# B&R Automation Studio project TD52 (part 126)

### Module_IC.var - Module global variables
```iecst
VAR
	ucEnergLev : USINT; (* ignition system energy level % *)
	ActTiming : INT; (* actual ignition timing 1/10 degree *)
	AdvTimLi : INT; (* advanced ingnition timing 1/10 deg *)
	AnzSPnt : USINT; (* number of ignition speed points *)
	AvgTim : SINT; (* average ignition timing 1/10 deg. *)
	bGnlTrip : BOOL;
	bGnlTrip1 : BOOL;
	bGnlTrip2 : BOOL;
	bGnlTrip3 : BOOL;
	bGnlWarning : BOOL;
	bInitOK : BOOL;
	bSelfTestOn : BOOL; (* TRUE= ignition is in sleftest mode *)
	bSpeedTrig2 : BOOL; (* TRUE=inverse speed trig 2 output *)
	BWS_HA : BOOL := 0; (* Betriebswahlschalter Hand/Auto *)
	CMSIgn_Init : CMSinit;
	CMSmain_Ign : CMSmain;
	ConfigIC : USINT; (* ignition system operating mode *)
	EnergLev : USINT; (* ignition system energy level in % *)
	E_Conf : ARRAY[0..38] OF USINT; (* event ignition system parameter *)
	E_IgnErr : USINT; (* events igniton system error *)
	E_IgnHW : USINT; (* events ignition system hardware *)
	E_IgnStat : USINT; (* events igniton system status *)
	E_Missf : ARRAY[0..2] OF USINT; (* events for misfire control *)
	E_SpeedUpd : USINT; (* event for ign. speed update time *)
	E_Timing : ARRAY[0..24] OF USINT; (* events ign. syetem indiv. timing *)
	E_ZDGSpeed : USINT; (* events for ignition engine speed *)
	FGDRPS : BOOL; (* Freigabe durch RPS *)
	FireOrder : ARRAY[0..24] OF USINT; (* engine ignition fire order *)
	GloTiPnt : INT; (* global timing point 1/10 degree *)
	GoSelftest : BOOL; (* switch ignition system to selftest *)
	ic900_vis : BOOL; (* TRUE=CAN ignition system is used *)
	iCylCount : USINT; (*Loop counter*)
	IC_Node : USINT; (* ignition system node number *)
	iECanDevGo : DINT;
	IgnErr : ARRAY[0..7] OF USINT; (* ignition system error messages *)
	IgnHW : ARRAY[0..7] OF USINT; (* ignition system hardware info *)
	IgnOFail : ARRAY[0..24] OF BOOL; (* ignition system cyl.output failure *)
	IgnStat : ARRAY[0..6] OF USINT; (* ignition system status info *)
	IgnVers : UINT; (* ignition system software version *)
	IndivTim : ARRAY[0..24] OF SINT; (* cylinder individual timing offset *)
	IN_IC : IN_IC_Struct := (0);
	MissfCmd : BOOL; (* command for start misfire *)
	MissfCyl : UDINT; (* cylinder misfire parameter *)
	MissfTim : UINT; (* misfire time parameter *)
	MM2VIS : MM2VIS_Struct;
	ModeIC : USINT; (* ignition system operating mode *)
	M_AGFD : BOOL := 0; (* Aggregat angefordert *)
	n_ist : INT; (* actual speed [1/min] *)
	OutFailR : USINT; (* ignition output failure rate para. *)
	OUT_IC : OUT_IC_Struct := (0);
	OvrSpeed : UINT; (* ignition overspeed parameter *)
	Para : PARA_IC_Struct;
	ParaFactoryDefault : PARA_IC_Struct := (0);
	pm : PARA_IC_Struct;
	PosResetIC : INT; (* ignition reset pickup position *)
	PROBE : BOOL := 0; (* Betriebsart PROBE *)
	QUITTRPS : BOOL := 0; (* ack comand to PLC-part *)
	RetTimLi : INT; (* ignition retard timing limit *)
	SecSpeed : UINT; (* ignition system security speed *)
	SecSpeedOld : UINT; (* last security speed value *)
	SpeedHys1 : UINT; (* hysteresis ign. speed trigger 1 *)
	SpeedHys2 : UINT; (* hysteresis ign. speed trigger 2 *)
	SpeedPnt : ARRAY[0..4] OF UINT; (* ignition timing speed points *)
	SpeedTrg2 : INT; (* ignition system speed trigger 2 *)
	SpeedTrig1 : INT; (* ignition system speed trigger 1 *)
	SpeedTrig2 : INT; (* ignition system speed trigger 2 *)
	SpeedUpd : UINT; (* ignition speed update time [ms] *)
	StopM : BOOL; (* TRUE=engine is stopped *)
	TimeSPnt : ARRAY[0..4] OF INT; (* ignition speed point timing *)
	TimingSeq : USINT; (* ignition system timing sequence *)
	ucIC900CommErrCount : USINT; (* comm. error counter *)
	ucIgnType : USINT; (* ignition system hardware type *)
	ucOutpFRate : USINT; (* ignition output failure rate para. *)
	ucZuendabst : USINT; (* ignition timing diff. row A to B *)
	ucZylZAus : USINT; (* cyl.inder with output failure *)
	usActSpeed : UINT; (* actual engine speed by ignition *)
	usIgnSystem : UINT; (* hardware type of ignition system *)
	usZahnzahl : UINT; (* number of starter ring gear teeth *)
	W_ZZP : INT; (* actual ignition timing setpoint *)
	xEngtype : EngType; (*FB for engine type specific values*)
	xOpMode : OpMode; (*FB for engine operation mode*)
	ZDGAUS : ARRAY[0..24] OF BOOL := [25(0)]; (*Ignition output monitoring*)
	ZDGAUS_A : BOOL; (*Ignition output monitoring*)
	ZDGAUS_B : BOOL; (*Ignition output monitoring*)
	ZDGAUS_W : BOOL; (*Ignition output monitoring*)
	ZDGCAM : BOOL := 0; (* ZDG AUSFALL CAM PICKUP *)
	ZDGCAN : BOOL := 0; (*Ignition CAN communication failure*)
	ZDGCPU : BOOL := 0; (* ZDG CPU FEHLER *)
	ZDGFALSCH : BOOL := 0; (*Wrong type of ignition system*)
	ZDGPAR : BOOL := 0; (* ZDG PARAMETRIERUNG IM BETRIEB *)
	ZDGPARAM : BOOL := 0; (* ZDG PARAMETER FEHLER *)
	ZDGRST : BOOL := 0; (* ZDG AUSFALL RESET PICKUP *)
	ZDGSpeed : tZDGSpeed; (* engine speed meassured by ignition *)
	ZDGTRI : BOOL := 0; (* ZDG AUSFALL TRIGGER PICKUP *)
	ZDGUEDZ : BOOL := 0; (*Ignition shutoff overspeed*)
	ZUEND : BOOL := 0; (*Ignition on*)
	ZylZahl : USINT;
	ZZPAvg : INT; (* actual ignition point average *)
	ZZPCyl : ARRAY[0..24] OF INT; (* actual cylinder igniton point *)
	ZZPMax : INT; (* actual max.cylinder ignition point *)
	ZZPMin : INT; (* actual min.cylinder ignition point *)
	zzp_ist : INT; (* aktuelle Soll-ZZP ohne Reduktion *)
	bNoInitDetected : BOOL := FALSE; (*allways true, except 1cycle on init up*)
	CMSmainTrigger : BOOL := FALSE; (*Trigger variable for CMS_main()*)
	SIM_rN_IgnIC_Act : REAL; (*WINMOD simulation: Engine speed measured by ignition IC*)
	iNum_ICSys : USINT; (*IC-System*)
	tIC_FiringDist : IC_FiringDist; (*Firing distances*)
	tIC_Curr : ARRAY[0..6] OF IC_Curr; (*Ignition pulse current and duration*)
	tIC_CoilPara : IC_CoilPara; (*General coil parameters*)
	tIC_SpDur : IC_SpDur; (*Spark duration*)
	tIC_SpdST : IC_SpdST; (*Self-test speed and speed ramp up / down time*)
	iTi_ICOn : UINT; (*Hours powered-up [h]*)
	tIC_U_Pickups : IC_U_Pickups; (*Pickup peak voltages*)
	iNum_PUMode : USINT; (*Pickup mode detected by SEMIC*)
	iNum_IC_SPAxSpdCoeff : UINT; (*SPAx speed coefficient A*)
	E_Global : ARRAY[0..21] OF USINT; (*Even variables for ignition global parameters*)
	tIC_SpInfo : ARRAY[0..24] OF IC_SpInfo; (*Spark voltage and primary energy demand*)
	E_IC_SpInfo : ARRAY[0..24] OF USINT; (*Event variables for spark voltage and primary energy demand*)
	iNum_IC_NrTeethErr : UINT; (*Number of teeth at pickup error*)
	E_IC_NrTeethErr : USINT; (*Event variable for number of teeth at pickup error*)
	iT_IC : INT; (*Ignition controller temperature [degC*10]*)
	E_T_IC : USINT; (*Event variable for ignition controller temperature*)
	iU_IC_Supply : INT; (*Ignition controller supply voltage [V*10]*)
	E_U_IC_Supply : USINT; (*Event variable for ignition controller supply voltage*)
	tIC_PUNoiseRate : IC_PUNoiseRate; (*Pickup noise rate*)
	E_IC_PUNoiseRate : USINT; (*Event variable for pickup noise rate*)
	tIC_PrimEnergyStat : IC_PrimEnergyStat; (*Minimum, maximum and average of the primary coil energy demand*)
	E_IC_PrimEnergyStat : USINT; (*Event variable for the minimum, maximum and average of the primary coil energy demand*)
	bB_TrigFail : BOOL; (*Operating message - Ignition failure trigger pickup*)
	bW_CamFail : BOOL; (*Warning - Ignition failure cam pickup*)
	bW_ResetFail : BOOL; (*Warning - Ignition failure reset pickup*)
	bW_TrigFail : BOOL; (*Warning - Ignition failure trigger pickup*)
	iNum_TrigFail : USINT; (*Operating message - Ignition failure trigger pickup - Indication*)
	tCoilParam : ARRAY[0..4] OF CoilParam; (*Coil parameters*)
	tCoilParam5 : CoilParam5; (*Coil parameters*)
	tCoilParam6 : CoilParam6; (*Coil parameters*)
	iNum_IC_Curr7 : UINT; (*Ignition pulse 7 current*)
	iTi_IC_IonTime : UINT; (*Ionization time [us]*)
	bW_IC_WrongFw : BOOL; (*Wrong ignition controller firmware*)
	iE_PrimEnergy_Min : UINT; (*Minimum primary energy demand [mJ]*)
	iE_PrimEnergy_Max : UINT; (*Maximum primary energy demand [mJ]*)
	iE_PrimEnergy_Avg : UINT; (*Average primary energy demand [mJ]*)
	bW_PUDegrad : BOOL; (*Warning - Pickup degradation*)
	VIS2MM : VIS2MM_Struct;
	bIC_BlockUpd : BOOL; (*Block engine stat during ignition controler firmware update*)
	bW_IC_Uin_Lo : BOOL; (*Warning - Ignition controller input voltage too low*)
	bA_IC_HwFail : BOOL; (*Alarm - Ignition controller hardware failure*)
	bSEMIC_Comm : BOOL; (*SEMIC CAN communication is active*)
	bW_PUWrongPol : BOOL; (*Wrong pickup polarity*)
	bA_WrongCoil : BOOL; (*Alarm - Wrong or missing ignition coil*)
	bB_WrongCoil : BOOL; (*Operating message - Wrong or missing ignition coil*)
	iNum_WrongCoil : USINT; (*Operating message - Wrong or missing ignition coil - Cylinder number*)
	bA_IC_CoilFail : BOOL; (*Alarm - Ignition coil or wiring failure*)
END_VAR
```

### Module_ICPara.typ - Module global parameter
```iecst
TYPE
	PROGRAMMER_INFO : 	STRUCT
		DO_NOT_SORT_PARA : STRING[40] := 'DO NOT CHANGE PARAMETER SORTING!'; (*DO NOT CHANGE PARAMETER SORTING!*) (*ADD NEW PARAMETER ONLY AT THE END OF THE Para STRUCTURE. DO NOT DELETE existing Para items.*)
	END_STRUCT;
	PARA_IC_Struct : 	STRUCT
		iEng_Motortype : INT; (*PARA: engine motortype*) (*OldName:motortyp; Cycle:;*)
		rCA_AdvTimeLim : REAL; (*PARA [12065]: advanced ignition timing 1/10 deg *) (*OldName:AdvTimLi; Cycle:;*)
		b_IgnIC_SpdTrig2Inv : BOOL; (*PARA [12053]: TRUE=inverse speed trig 2 output *) (*OldName:bSpeedTrig2; Cycle:;*)
		rIgnIC_PowLev : REAL; (*PARA [12056]: ignition system energy level in % *) (*OldName:EnergLev; Cycle:;*)
		b_IgnIC_900Active : BOOL; (*PARA [12062]: TRUE=CAN ignition system is used *) (*OldName:ic900_vis; Cycle:;*)
		r_IgnIC_OutpMon : REAL; (*PARA [12054]: ignition output failure rate para. *) (*OldName:OutFailR; Cycle:;*)
		rN_OvrSpeed : REAL; (*PARA [12129]: Ignition overspeed limit*) (*OldName:OvrSpeed; Cycle:;*)
		r_IgnIC_ResPosIC : REAL; (*PARA [12055]: ignition reset pickup position *) (*OldName:r_IgnIC_ResPosIC; Cycle:;*)
		rCA_RetTimeLim : REAL; (*PARA [12066]: ignition retard timing limit *) (*OldName:RetTimLi; Cycle:;*)
		rN_IgnIC_SecSpeed : REAL; (*PARA [12059]: ignition system security speed *) (*OldName:SecSpeed; Cycle:;*)
		rN_IgnIC_HySpeed1 : REAL; (*PARA [12057]: hysteresis ign. speed trigger 1 *) (*OldName:SpeedHys1; Cycle:;*)
		rN_IgnIC_HySpeed2 : REAL; (*PARA [12058]: hysteresis ign. speed trigger 2 *) (*OldName:SpeedHys2; Cycle:;*)
		rN_IgnIC_SpeedTrig1 : REAL; (*PARA [12060]: ignition system speed trigger 1 *) (*OldName:SpeedTrig1; Cycle:;*)
		rN_IgnIC_SpeedTrig2 : REAL; (*PARA [12061]: ignition system speed trigger 2 *) (*OldName:SpeedTrig2; Cycle:;*)
		zz_V4_0_ParaVersionEnd : REAL := 4.0; (*! ADD NEW PARAMETER ONLY BELOW THIS LINE ! This is the end of base version parameter and has to stay unchanged. DO NOT CHANGE SORT ORDER of Para!*) (* OldName: new PV; Cycle: 5; *)
		bSEMIC_Active : BOOL; (*PARA[14519]: Ignition controller SEMIC*)
		rNum_IC_RelFwVer : REAL; (*PARA[14520]: Released SEMIC firmware version*)
		iNum_IC_PUMode : USINT; (*PARA[14521]: Pickup mode*)
		iNum_IC_CoilType : USINT; (*PARA[14522]: SEMIC coil type*)
		iTi_IC_TimeToPeak : UINT; (*PARA[14523]: Time to peak voltage [us]*)
		iI_IC_CoilCurrMax : USINT; (*PARA[14524]: Maximum primary coil current [A]*)
		iNum_IC_IgnEnergyMax : UINT; (*PARA[14525]: Maximum energy for firing event [mJ]*)
		iSpd_IC_PUMon : UINT; (*PARA[14526]: Speed to activate pickup monitoring [rpm]*)
		rU_IC_PUMin : REAL; (*PARA[14527]: Minimum pickup voltage [V]*)
		rSA_SparkDuration : REAL; (*PARA [12152]: SAFI spark duration  *)
		rSA_DurTol : REAL; (*PARA [12134]: spark duration deviation limit *) (* OldName:ucDurTol; Cycle: *)
		rSA_SparkCurChar : REAL; (*PARA [12150]: spark current characteristic*)
		rSA_SparkCurLev : REAL; (*PARA [12151]: spark current level *) (* OldName:ucSparkCurLev; Cycle: *)
		bDynSparkDuration : BOOL; (*PARA [13646]: Variable spark duration active *) (* OldName:newPV; Cycle: *)
		rP_Act_DynSpark_Limit_Nom : REAL; (*PARA [13648]: Spark duration below power threshold *) (* OldName:newPV; Cycle: *)
		usDurationIdle : UINT; (*PARA [13647]: Spark duration below power threshold *) (* OldName:newPV; Cycle: *)
		tSA_Ign_0 : IC_CurrPmmReal; (*PARA [12165]: SAFI ionization duration*) (* OldName:SAFICurr0PMM; Cycle: *)
		tSA_Ign_1 : IC_CurrPmmReal; (*PARA [12166] & PARA [12167] SAFI ignition current / duration setting 1 *) (* OldName:SAFICurr1PMM; Cycle: *)
		tSA_Ign_2 : IC_CurrPmmReal; (*PARA [12168] & PARA [12169]: SAFI ignition current / duration setting 2 *) (* OldName:SAFICurr2PMM; Cycle: *)
		tSA_Ign_3 : IC_CurrPmmReal; (*PARA [12170] & PARA [12171]: SAFI ignition current / duration setting 3 *) (* OldName:SAFICurr3PMM; Cycle: *)
		tSA_Ign_4 : IC_CurrPmmReal; (*PARA [12172] & PARA [12173]: SAFI ignition current / duration setting 4 *) (* OldName:SAFICurr4PMM; Cycle: *)
		tSA_Ign_5 : IC_CurrPmmReal; (*PARA [12174] & PARA [12175]: SAFI ignition current / duration setting 5 *) (* OldName:SAFICurr5PMM; Cycle: *)
		tSA_Ign_6 : IC_CurrPmmReal; (*PARA [12176]: SAFI ignition current setting 6 *) (* OldName:SAFICurr6PMM; Cycle: *)
		rNum_IC_TPCSCx1 : REAL; (*PARA[14528]: Breakpoint of secondary current axis for the target primary current 2D-MAP - X1*)
		rNum_IC_TPCSCx2 : REAL; (*PARA[14529]: Breakpoint of secondary current axis for the target primary current 2D-MAP - X2*)
		rNum_IC_TPCSCx3 : REAL; (*PARA[14530]: Breakpoint of secondary current axis for the target primary current 2D-MAP - X3*)
		rNum_IC_TPCSCx4 : REAL; (*PARA[14531]: Breakpoint of secondary current axis for the target primary current 2D-MAP - X4*)
		iNum_IC_TPCAPVy1 : USINT; (*PARA[14532]: Breakpoint of accumulated primary voltage axis for the target primary current 2D-MAP - Y1*)
		iNum_IC_TPCAPVy2 : USINT; (*PARA[14533]: Breakpoint of accumulated primary voltage axis for the target primary current 2D-MAP - Y2*)
		iNum_IC_TPCAPVy3 : USINT; (*PARA[14534]: Breakpoint of accumulated primary voltage axis for the target primary current 2D-MAP - Y3*)
		iNum_IC_TPCAPVy4 : USINT; (*PARA[14535]: Breakpoint of accumulated primary voltage axis for the target primary current 2D-MAP - Y4*)
		iI_IC_TPCx1y1 : USINT; (*PARA[14536]: Target primary current 2D-MAP data point - X1Y1*)
		iI_IC_TPCx1y2 : USINT; (*PARA[14537]: Target primary current 2D-MAP data point - X1Y2*)
		iI_IC_TPCx1y3 : USINT; (*PARA[14538]: Target primary current 2D-MAP data point - X1Y3*)
		iI_IC_TPCx1y4 : USINT; (*PARA[14539]: Target primary current 2D-MAP data point - X1Y4*)
		iI_IC_TPCx2y1 : USINT; (*PARA[14540]: Target primary current 2D-MAP data point - X2Y1*)
		iI_IC_TPCx2y2 : USINT; (*PARA[14541]: Target primary current 2D-MAP data point - X2Y2*)
		iI_IC_TPCx2y3 : USINT; (*PARA[14542]: Target primary current 2D-MAP data point - X2Y3*)
		iI_IC_TPCx2y4 : USINT; (*PARA[14543]: Target primary current 2D-MAP data point - X2Y4*)
		iI_IC_TPCx3y1 : USINT; (*PARA[14544]: Target primary current 2D-MAP data point - X3Y1*)
		iI_IC_TPCx3y2 : USINT; (*PARA[14545]: Target primary current 2D-MAP data point - X3Y2*)
		iI_IC_TPCx3y3 : USINT; (*PARA[14546]: Target primary current 2D-MAP data point - X3Y3*)
		iI_IC_TPCx3y4 : USINT; (*PARA[14547]: Target primary current 2D-MAP data point - X3Y4*)
		iI_IC_TPCx4y1 : USINT; (*PARA[14548]: Target primary current 2D-MAP data point - X4Y1*)
		iI_IC_TPCx4y2 : USINT; (*PARA[14549]: Target primary current 2D-MAP data point - X4Y2*)
		iI_IC_TPCx4y3 : USINT; (*PARA[14550]: Target primary current 2D-MAP data point - X4Y3*)
		iI_IC_TPCx4y4 : USINT; (*PARA[14551]: Target primary current 2D-MAP data point - X4Y4*)
		rNum_IC_PVOTRPCx1 : REAL; (*PARA[14552]: Breakpoint of spark current axis for the primary voltage off time reference 1D-TABLE - X1*)
		rNum_IC_PVOTRPCx2 : REAL; (*PARA[14553]: Breakpoint of spark current axis for the primary voltage off time reference 1D-TABLE - X2*)
		rNum_IC_PVOTRPCx3 : REAL; (*PARA[14554]: Breakpoint of spark current axis for the primary voltage off time reference 1D-TABLE - X3*)
		rNum_IC_PVOTRPCx4 : REAL; (*PARA[14555]: Breakpoint of spark current axis for the primary voltage off time reference 1D-TABLE - X4*)
		rNum_IC_PVOTRPCx5 : REAL; (*PARA[14556]: Breakpoint of spark current axis for the primary voltage off time reference 1D-TABLE - X5*)
		rNum_IC_PVOTRx1 : REAL; (*PARA[14557]: Duty cycle reference 1D-TABLE data point - X1*)
		rNum_IC_PVOTRx2 : REAL; (*PARA[14558]: Duty cycle reference 1D-TABLE data point - X2*)
		rNum_IC_PVOTRx3 : REAL; (*PARA[14559]: Duty cycle reference 1D-TABLE data point- X3*)
		rNum_IC_PVOTRx4 : REAL; (*PARA[14560]: Duty cycle reference 1D-TABLE data point- X4*)
		rNum_IC_PVOTRx5 : REAL; (*PARA[14561]: Duty cycle reference 1D-TABLE data point- X5*)
		iNum_IC_APVCF : USINT; (*PARA[14562]: Accumulated primary voltage compensation factor. Used for target primary current compensation for non nominal secondary voltage*)
		iI_IC_MPCPVOff : USINT; (*PARA[14617]: Calibration parameter for spark diagnostics. Minimum primary current after 250us spark duration if no 80v is applied*)
		iI_IC_MPCPVOn : USINT; (*PARA[14618]: Calibration parameter for spark diagnostics. Minimum primary current after 250us spark duration if 80v is applied for 250us*)
	END_STRUCT;
END_TYPE
```

### Program Logical/ICxx/IN_IC (IEC, version 4.12.0) - + IN-Task

- IN_ICCyclic.st (not readable text: treated as protected, skipped)

#### IN_IC.var - Local variables
```iecst
VAR
	iNum_IC_SpCurChar : USINT; (*Spark characteristic selection*)
	iNum_IC_SpCurLvl : USINT; (*Spark current level [%]*)
	iNum_IC_SpCurCharOld : USINT; (*Old spark characteristic selection*)
	iNum_IC_SpCurData : ARRAY[0..10] OF UINT; (*Data from IC_Curr.dat*)
	xDatObjRead_ICxxCurr : DatObjRead; (*FuB to read the data from IC_Curr.dat*)
	tIC_CurrPMM : ARRAY[0..7] OF IC_Curr; (*Ignition pulse current and duration from the parameters*)
	xDatObjInfo_ICxxCurr : DatObjInfo; (*FuB to read the info from IC_Curr.dat*)
	xDatObjInfo_ICxxCoil : DatObjInfo; (*FuB to read the info from IC_Coil.dat*)
	xDatObjRead_ICxxCoil : DatObjRead; (*FuB to read the data from IC_Coil.dat*)
	iNum_IC_CoilType : USINT; (*Coil type*)
	iNum_IC_CoilTypeOld : USINT; (*Old coil type*)
	iNum_IC_SpCoilData : ARRAY[0..39] OF UINT; (*Data from IC_Coil.dat*)
END_VAR
```

### Program Logical/ICxx/OUT_IC (IEC, version 4.14.0) - + OUT-Task

- OUT_ICCyclic.st (not readable text: treated as protected, skipped)

#### OUT_IC.var
```iecst
VAR
	xTON_IgnEngergy_Hi : TON; (*Timer for warning maximum energy exceeded*)
END_VAR
```

### Program Logical/ICxx/ignition (IEC, version 4.13.0) - + Main igniton task 

- ignitionCyclic.st (not readable text: treated as protected, skipped)

- ignitionInit.st (not readable text: treated as protected, skipped)

#### ignition.var
```iecst
VAR
	ucStateOfPar : USINT; (* state of parameter transmission *)
	bIC900Comm : BOOL; (* TRUE=communication to ignition OK *)
	bIgnOK : BOOL; (* TRUE=ignition system is OK *)
	bIgnFire : BOOL; (* TRUE=ignition system is firing *)
	bSendIC900Par : BOOL; (* flag sending ignition parameter *)
	bSendRunPar : BOOL; (* falg sending igniton run parameter *)
	bSendRunParError : BOOL; (* TRUE=error send ignition run para. *)
	bSendIC900ParError : BOOL; (* TRUE=error send igniton parameter *)
	bResetIC900 : BOOL; (* flag for reseting ignition system *)
	bChangeBetrArt : BOOL; (* TRUE=change ignition operating mod *)
	bChangeBTRFailure : BOOL; (* TRUE=fault change operating mode *)
	ucIgnOFailTimer : ARRAY[0..24] OF USINT; (* ignition output failure timer *)
	ucZylCount : USINT; (* cylinder loop counter *)
	ucModeIC : USINT; (* igniton system operating mode *)
	ucTimingSeq : USINT; (* ingition system timing sequence *)
	ucResetState : USINT; (* state of igniton reset sequence *)
	ucIC900Hours : UINT; (* ignition system operating hours *)
	usZahnzahlOld : UINT; (* number of starter ring gear teeth *)
	usSelfTestOnTime : UINT; (* timer for selftest on time *)
	bIC900Off : BOOL; (* TRUE=stop comm. to ignition system *)
	ssZZPMin : INT; (* actual min. indiv. timing point *)
	ssZZPMax : INT; (* actual max. indiv. timing point *)
	TON_ZDGTRI : TON; (* delay error missing ring gear *)
	F_TRIG_ZUEND : F_TRIG; (* faling trigger ignition system on *)
	R_TRIG_EngQuitt : R_TRIG; (* FUB trigger alarm reset pushed *)
	R_TRIG_EngStop : R_TRIG; (* FUB trigger operating switch stop *)
	R_TRIG_EngDemand : R_TRIG; (* FUB trigger for engine demand *)
	ucStateOfChange : USINT; (* state of change operating mode *)
	TON_ZDGRST : TON; (* FUB delay reset signal missing *)
	TON_ZDGPARAM : TON; (* FUB delay no config at enabele run *)
	TON_ZDGCAM : TON; (* FUB delay camshaft signal missing *)
	TON_BTRTimeOut : TON; (* 1 sec. timeout for sending IC mode *)
	ucIgnParCount : USINT; (* parameter error counter *)
	ucStateIgnPar : USINT; (* state of ignition parameter send *)
	bSendIgnParError : BOOL; (* TRUE=error send ignition parameter *)
	ucIndivTimCnt : USINT; (* loop counter individual timing *)
	PosResetICOld : INT; (* last ignition reset pickup pos. *)
	OutFailROld : USINT; (* last ign. outp. faulure rate para. *)
	AdvTimLiOld : INT; (* lat advanced timing limit *)
	RetTimLiOld : INT; (* last retard timing limit *)
	OvrSpeedOld : UINT; (* last over speed value *)
	SpeedTrig1Old : INT; (* last speed trigger 1 value *)
	SpeedTrig2Old : INT; (* last speed trigger 2 value *)
	SpeedHys1Old : UINT; (* last speed hystersis 1 value *)
	SpeedHys2Old : UINT; (* last speed hystersis 2 value *)
	TON_SecondTick : TON; (* second tick TRUE for 0,1 sec. *)
	ucNrOfZDGAUS : USINT; (* number of ign. output failures *)
	AmmSeqZDGAUS : AmmSequence; (* FUB AmmSequence ign. output fail. *)
	bSEMIC_ICmode : BOOL; (*SEMIC in IC-mode*)
	bIC_PUmodeRead : BOOL; (*PU mode read at least once since the CAN communication was open*)
END_VAR
```

### Program Logical/ICxx/SpeedIC (IEC, version 4.13.0) - + Engine speed ignition system IC

- SpeedICCyclic.st (not readable text: treated as protected, skipped)

#### SpeedIC.var - Local variables
```iecst
VAR
	MissfCyl_Old : UDINT;
	bIC_MissfCmd_Old : BOOL; (*Command to start skip fire - old*)
	xTOF_MissfCmd : TOF; (*Delay to turn off the skip fire command*)
END_VAR
```

### Program Logical/ICxx/ICGen (IEC, version 4.14.0) - + Task for general issues 

- GeneralCyclic.st (not readable text: treated as protected, skipped)

### Program Logical/ICxx/SEMIC (IEC, version 4.14.0) - + SEMIC ignition task

- SEMICCyclic.st (not readable text: treated as protected, skipped)

- SEMICInit.st (not readable text: treated as protected, skipped)

#### SEMIC.var - Local variables
```iecst
VAR CONSTANT
	all : SINT := 127;
	none : SINT := -1;
END_VAR
VAR
	bAmmSeqClkP : BOOL; (*Clock for AmmSequence*)
	bIC_RE_EngStop : BOOL; (*Rising edge of engine stopped + 5 s*)
	bIC_RE_SwReset : BOOL; (*Rising edge of the alarm reset button at engine stand still*)
	bIN_WrongFw : BOOL; (*Input of timer for alarm Wrong ignition controller firmware*)
	bSEMIC_CfgNotAllow : BOOL; (*Configuration parameters tranfer not allowed if engine is running*)
	bSEMIC_IgnFire : BOOL; (*Ignition firing*)
	bSEMIC_IgnOK : BOOL; (*Ignition OK*)
	bSEMIC_OpBeforeCfg : BOOL; (*Send operation data before the configuration data*)
	bSEMIC_SelfTestStart : BOOL; (*Start self test procedure for SEMIC*)
	bSEMIC_SelfTestStop : BOOL; (*Stop self test procedure for SEMIC*)
	bSEMIC_SendAllOpData : BOOL; (*Trigger the sending of all operating data*)
	bSEMIC_SendConfig : BOOL; (*Activate sending of configuration data*)
	bSEMIC_SwReset : BOOL; (*Start the SW reset procedure*)
	bToggle : BOOL;
	iCA_AdvTimLiOld : INT; (*Old advance timing limit*)
	iCA_ITPCyl : ARRAY[0..24] OF INT; (*Cylinder-specific ignition timing point difference from the global timing point*)
	iCA_PosResetICOld : INT; (*Old reset position*)
	iCA_RetTimLiOld : INT; (*Old retard timing limit*)
	iE_PrimEnergy_Sum : UDINT; (*Sum used to calculate the average primary coil energy demand*)
	iNum_Cnt : USINT;
	iNum_ConfigPara : SINT; (*Number of the configuration data to be sent*)
	iNum_ConfState : USINT; (*State of the configuration data sending sequence*)
	iNum_CylCnt : USINT;
	iNum_EnergLevOld : USINT; (*Old energy level*)
	iNum_GlobalPara : USINT; (*Number of the operating data to be sent*)
	iNum_ICSysOld : USINT; (*Old IC-system*)
	iNum_IC_Curr7Old : UINT; (*Old ignition pulse 7 current*)
	iNum_IC_SPAxSpdCoeffOld : UINT; (*Old SPAx speed coefficient A*)
	iNum_OutFailROld : USINT; (*Old output failure rate*)
	iNum_ParaCnt : USINT;
	iNum_ReadVarCnt : USINT; (*Counter for the variable read requests sequencing*)
	iNum_ReSendCnt : USINT;
	iNum_ResetState : USINT;
	iNum_SelfTestState : USINT;
	iNum_StartComCnt : USINT;
	iNum_TimingSeqOld : USINT; (*Old timing sequence*)
	iNum_ZahnzahlOld : UINT; (*Old number of gear teeth*)
	iNum_ZylZahlOld : USINT; (*Old number of cylinders*)
	iN_ActSpeed : UINT; (*Actual speed*)
	iN_OvrSpeedOld : UINT; (*Old overspeed*)
	iN_SpeedHys1Old : UINT; (*Old hysteresis speed trigger 1*)
	iN_SpeedHys2Old : UINT; (*Old hysteresis speed trigger 2*)
	iN_SpeedTrig1Old : INT; (*Old speed trigger 1*)
	iN_SpeedTrig2Old : INT; (*Old speed trigger 2*)
	iTi_IC_IonTimeOld : UINT; (*Old ionization time*)
	iTi_MissfTimOld : UINT; (*Old maximum skip fire duration*)
	iTi_SpeedUpdOld : UINT; (*Old speed update time*)
	tCoilParam5Old : CoilParam5; (*Old coil parameters*)
	tCoilParam6Old : CoilParam6; (*Old coil parameters*)
	tCoilParamOld : ARRAY[0..4] OF CoilParam; (*Old coil parameters*)
	tIC_CoilParaOld : IC_CoilPara; (*Old general coil parameters*)
	tIC_CurrOld : ARRAY[0..6] OF IC_Curr; (*Old ignition pulse current and duration*)
	tIC_FiringDistOld : IC_FiringDist; (*Old firing distances*)
	tIC_SpdSTOld : IC_SpdST; (*Old self-test speed and speed ramp up/down time*)
	tIC_SpDurOld : IC_SpDur; (*Old spark duration*)
	xAmmSeqIgnOFail : AmmSequence; (*Alarm sequence for Ignition output monitoring*)
	xAmmSeqWrongCoil : AmmSequence; (*Alarm sequence for Wrong or missing ignition coil*)
	xTON_100msTick : TON; (*100ms based clock pulse*)
	xTON_bW_TrigFail : TON; (*Timer for Warning - Ignition failure trigger pickup*)
	xTON_ConfFail : TON; (*Timer for configuration state too long*)
	xTON_EngineStop : TON; (*Timer for SEMIC software reset*)
	xTON_IcNoOpState : TON; (*Timer for Ignition parameter error if engine is demanded and IC is not in operation state*)
	xTON_IC_WrongFw : TON; (*Timer for alarm Wrong ignition controller firmware*)
	xTON_IgnDemFall : TON; (*Falling edge of the ignition demand*)
	xTON_IgnDemRise : TON; (*Rising edge of the ignition demand*)
	xTON_ResetFail : TON; (*Timer for ignition controller software reset too long*)
	xTON_SecondTick : TON; (*1s based clock pulse*)
	xTON_ZDGCAM : TON; (*Timer for Ignition failure cam pickup*)
	xTON_ZDGPARAM : TON; (*Timer for re-parametrization because of parametrization failure*)
	xTON_ZDGRST : TON; (*Timer for Ignition failure reset pickup*)
	xTON_ZDGTRI : TON; (*Timer for Alarm - Ignition failure trigger pickup*)
	xTON_ZDGTRI_4PU : TON; (*Timer for Alarm - Ignition failure trigger pickup in 4-pickups mode*)
	xTON_ZDGTRI_NoFire : TON; (*Timer for Alarm - Ignition failure trigger pickup when ignition not firing*)
END_VAR
```

### Program Logical/ICxx/MsgIC (IEC, version 4.13.0) - + Messages

- MsgICCyclic.st (not readable text: treated as protected, skipped)

- MsgICInit.st (not readable text: treated as protected, skipped)

#### MsgIC.var - Local variables
```iecst
VAR
	iAdrAmmBase2MM : UDINT;
	iAdrMM2AmmBase : UDINT;
	xMsg3310 : Msg;
	xMsg3240 : Msg;
	xMsg3410 : Msg;
	xMsg3027 : Msg;
	xMsg3031 : Msg;
	xMsg3029 : Msg;
	xMsg3030 : Msg;
	xMsg3026 : Msg;
	xMsg3025 : Msg;
	xMsg3028 : Msg;
	xMsg3052 : Msg;
	xMsg3209 : Msg;
	xMsg9339 : Msg;
	xMsg9340 : Msg;
	xMsg9049 : Msg;
	xMsg9341 : Msg;
	xMsg9342 : Msg;
	xMsg9343 : Msg;
	xMsg9315 : Msg;
	xMsg2363 : Msg;
	xMsg2764 : Msg;
	xMsg2767 : Msg;
	xMsg2367 : Msg;
	xMsg9073 : Msg;
	xMsg2375 : Msg;
END_VAR
```

### Program Logical/ICxx/ParIC (IEC, version 4.06.0) - + Parameter handling

- perm_par.st (not readable text: treated as protected, skipped)

#### perm_par.var
```iecst
VAR
	tParaIntern : ParaHandler_typ; (*Connector type to perm_par*)
	tMM2ParaBase_ReadBack : MM2ParaBase_type; (*INTERNAL! V4.06 new readback structure for information from previous tasks*)
	bWriteDataObj : BOOL; (* TRUE=write data object module *)
	bDataObjLenErr : BOOL; (*Error occured in permem: data module size missmatch*)
	bCreateDataObj : BOOL; (* TRUE=create new data object *)
	bWriteOnce : BOOL; (* write permanent memory once *)
	DatObjCreate_01 : DatObjCreate; (* data object create *)
	DatObjInfoBak_02 : DatObjInfo; (* data object info *)
	DatObjDelete_01 : DatObjDelete; (* data object delete *)
	DatObjRead_01 : DatObjRead; (* data object read *)
	DatObjRead_02 : DatObjRead; (* manual initiated data object read *)
	DatObjWrite_01 : DatObjWrite; (* data object write *)
	DatObjDelete_02 : DatObjDelete; (* data object delete *)
	DatObjDelete_11 : DatObjDelete; (*Delete Backup File*)
	DatObjInfo_01 : DatObjInfo; (* data object info *)
	DatObjInfo_02 : DatObjInfo; (* data object info *)
	szModuleName : STRING[35]; (* module name of object *)
	szModuleNameBackup : STRING[35]; (* module name of posiibly created backup object *)
	DatObjCopy_01 : DatObjCopy;
	bCopyDataObj : BOOL;
	TON_WarnDelay : TON;
	TON_WritePMEM : TON; (* delay write permanent memory *)
	ulPMPointer : UDINT; (* adress of actual checksum value *)
	ulChecksum : UDINT; (* parameter checksum value *)
	pm_len : UDINT; (* permanent value lenght *)
	ulChecksumOld : UDINT; (* last vlaue of parameter checksum *)
	ulChkValue : UDINT; (* actual value of parameter pointer *)
	pm_id : UDINT; (* permanent value identifier *)
	pm_p : UDINT; (* permanent value pointer *)
	DatObjInfo_META : DatObjInfo;
	DatObjRead_META : DatObjRead;
	szMetaDataRaw : STRING[2000];
	szMetaData : ARRAY[0..4] OF STRING[35];
	szMetaDataVis : ARRAY[0..3] OF STRING[35];
	ssIndex : INT;
	ssCount : INT;
	ucMetaDataRaw : ARRAY[0..2000] OF USINT;
	ssCount2 : INT;
	szMetaDataFile : STRING[10];
	szText1 : STRING[20];
	pv_adr_IN_XX_tPB2MM : UDINT;
	pv_lng : UDINT;
	pv_lng_IN_XX_tPB2MM : UDINT;
	pv_lng_OUT_XX_tPB2MM : UDINT;
	szText2 : STRING[20];
	pv_adr_OUT_XX_tXX2PB : UDINT;
END_VAR
VAR CONSTANT
	ERR_NOERROR : UINT := 0;
END_VAR
VAR
	usPMWriteCnt : UINT;
	pm_Error : UDINT; (* permanent value error *) (* Deleted: pm : ParaMem_typ; permanent memory tags mathias, 22.8.11*)
	fun_Error : UDINT := 0; (*state > 0 = function error*)
	xLocalParaCheck : ParaCheckFUB; (*local function instance to check parameter values*)
	TON_ParaSetupOk : TON;
	bParaCheckSystemOk : BOOL;
	iDebug_ParaOkChecked : UDINT;
	bRestoreBackupDataObj : BOOL := FALSE;
	bRestoreDataObjContent : BOOL := FALSE;
	pm_id_backup : UDINT;
	pm_p_Backup : UDINT;
	DatObjCopy_02 : DatObjCopy;
	bDeleteBackupDataObj : BOOL := FALSE; (*Command to delete backup data module file on purpose*)
	bDebugPara : ARRAY[0..5] OF BOOL;
	ssIndex2 : INT;
	ssIndex3 : INT;
	ssIndex4 : INT;
	ssIndexVis : INT;
	szText : STRING[40];
	pv_adr_Para : UDINT;
	szParaSnippet : ARRAY[0..5] OF STRING[150];
	szParaIndex : STRING[10];
	slValue : DINT;
	iModuleDLD_ResetCount : INT;
	bDownloadDetected : BOOL;
	bFlagParaStructCopyWorking : BOOL; (*true, if cyclic para copying is active, 1 false cycle at every copy *)
	bStoreInitParaInDataObj : BOOL := FALSE;
	bTestflag : BOOL;
	bReadOutMETA_Once : BOOL;
	tParaCheck_iPvAdress : ARRAY[0..5] OF UDINT;
	tParaCheck_iPvLengt : ARRAY[0..5] OF UDINT;
	tParaCheck_rPvValue : ARRAY[0..5] OF REAL;
	tParaCheck_rRangeMIN : ARRAY[0..5] OF REAL;
	tParaCheck_rRangeMAX : ARRAY[0..5] OF REAL;
	tParaCheck_szPvName : ARRAY[0..5] OF STRING[35];
	ssFormatDetected : INT;
	szMetaDataPart : STRING[150];
	szFullTaskName : STRING[35];
	szFullMetaModuleName : STRING[35];
	debugLen : INT;
	debugSize : INT := 0;
	strcat_adr1 : UDINT;
	strcat_adr2 : UDINT;
	ssIndexTN : INT;
	bAlternate : BOOL;
	n : INT;
	iAlternateChecksum : DINT;
	iAlternateChecksumOld : DINT;
	ulDebugChkValue : ARRAY[0..999] OF UDINT;
	Adr1 : UDINT;
	Adr2 : UDINT;
	usPMWriteCntStepsize : UINT := 1; (*different step sizes to help debug*)
	usPMWriteCntXOR : UINT;
	usPMWriteCntAltSum : UINT;
	ulAdrPM : UDINT;
	usChkValuePM : USINT;
	ulAdrPara : UDINT;
	ulPara_len : UDINT;
	usChkValuePara : USINT;
	iDebugCountPMDifferences : DINT := 0;
	bEngineRunDetected : BOOL; (*detection status bit autocommand 100 /101  for engine run state*)
	ucMetaDataDebugInfoLine : ARRAY[0..24] OF STRING[80];
	ssIndexMand : INT := 0;
	szMetaDataMand : STRING[35];
	iMyErrorInfo_Autoreset : DINT; (*internal autoreset counter*)
	ssIndex_Version : INT; (*internal*)
	ssIndex_BU : INT; (*internal*)
	ssIndex_BU2 : INT; (*internal*)
END_VAR
```

### Program Logical/ICxx/VisIC (IEC, version 4.12.0) - + Visualization task

- VisICCyclic.st (not readable text: treated as protected, skipped)

#### VisIC.var - Local variables
```iecst
VAR
	iNum_CylCnt : USINT;
END_VAR
```

### Package Logical/ICxx/CAN - CAN communication IC

### Program Logical/ICxx/CAN/caniniIc (IEC, version 4.00.3) - + IC CAN communication init

#### caniniIcCyclic.st
```iecst
(*******************************************************************************
AGGR: intiate CAN communication (cyclic)

This code is confidential and proprietary to the INNIO Company.
It may not be used in any form, or reproduced in any manner, without the express
written permission of the INNIO Company.
Copyright, INNIO Company, 2022

Customized modifications: -
------------------------

History:
-------
V0.1		31-08-2001	Fahringer, generated from caninit.c V0.2
			31-08-2001	Fahringer, last modification
V0.21		14-10-2003	Weitzer,   transfer all CAN and CMS FUBs to caninit task
V0.40		14-02-2007  Weitzer,   change to new standard IF (SL1.SS1.IF2)
							   	   delete MMD (multimeasure device)
V0.50		07-09-2007	Weitzer,   SAFI added
							       main FUB´s moved to canmain program
V0.60		23-02-2010	Weitzer,   SAFI2 (prot injection) added
V4.00.03	10-07-2014	Denk,      AND ic900_vis added
V4.00.05	15-07-2015	Weitzer,   move CMS main Fub to SpeedIC task
V4.12.00	08-09-2022	Andre	   Select the engine speed from the ICxx module also if SEMIC is active

Instructions for use:
--------------------
-initiate the CAN-Bus communictation controller
-initiate CAN CMS manager

Outstandings:
------------
*******************************************************************************)

PROGRAM _CYCLIC

	IF IN_IC.iCANIdent <> 0 AND NOT bInitOK AND (ic900_vis OR Para.bSEMIC_Active) THEN	(* check if CAN open was successful *)

		(*initiate CMS manager Ignition *)
		CMSIgn_Init(enable:=1, us_ident:=IN_IC.iCANIdent, user_type:=0, queue_cnt:=0, modul_name:=ADR('cmsign'));
		(* initiate CMS main function for send and receive Ignition CAN messages *)
		CMSmain_Ign.enable    := TRUE;
		CMSmain_Ign.cms_ident := CMSIgn_Init.cms_ident;
		CMSmain_Ign.cms_mode  := 2;

		IF CMSIgn_Init.status = 0 THEN
			bInitOK := TRUE;
		END_IF
	END_IF

END_PROGRAM
```

### Data object Logical/ICxx/CAN/cmsign (Simple, version 4.12.0) - + IC CAL ignition

- cmsign.dat (binary file, 13439 bytes)
### Program Logical/ICxx/CAN/IC_Updater (IEC, version 4.13.0) - + IC CAN updater

- IC_UpdaterCyclic.st (not readable text: treated as protected, skipped)

- IC_UpdaterInit.st (not readable text: treated as protected, skipped)

#### IC_Updater.var - Local variables
```iecst
VAR
	bIC_StartFwUpd : BOOL; (*Start the IC firmware download*)
	CMSdlreq_IcFw : CMSdlreq; (*Function block to download IC firmware*)
	DatObjInfo_IcFw : DatObjInfo; (*Function block to get the info of the ICfirmware*)
	iNum_IcFwAdr : UDINT; (*IC firmware address*)
	iNum_IcFwLen : UDINT; (*IC firmware length*)
	iNum_IcFwStatus : UINT; (*IC firmware status*)
	iNum_IcUpdState : USINT;
	iNum_InitDlFwCnt : USINT; (*Counter to re-send the initiate domain download*)
	xTON_IC_Upd : TON; (*Limit the IC firmware download to 30 min*)
END_VAR
```

### Package Logical/ICxx/DataIC - Data ICxx

### Data object Logical/ICxx/DataIC/IC_Coil (Simple, version 4.12.0) - + IC coil type data

- IC_Coil.dat (binary file, 45687 bytes)
### Data object Logical/ICxx/DataIC/IC_Curr (Simple, version 4.12.0) - + IC spark current characteristic

- IC_Curr.dat (binary file, 12102 bytes)
### Package Logical/Ignition - IG: Ignition

### Data object Logical/Ignition/META_IG (Simple) - MODUL META data file

#### META_IG.dat
```
; *******************************************************************************
; AGGR: Module Meta Data (data module)
;
; This code is confidential and proprietary to the INNIO Company.
; It may not be used in any form, or reproduced in any manner, without the express
; written permission of the INNIO Company.
; Copyright, INNIO Company, 2025
;
; Customized modifications: -
; ------------------------
;
; History:
; -------
; V03.99.00.00	06.03.2013	Weitzer		generated for modular software
; V03.99.02.00	29.05.2013	Zengerer	initial dependencies prepared
; V04.00.00.00	30.01.2014	Denk		new version
; V04.01.00.00	22.07.2014	Denk		OUT_IG.rCA_Ign_Avg added, Para task updated, bIgn_SelfTest to MM2VIS added
; V04.03.00.00	02.11.2015	Zengerer 	MANDATORYMODULE statement
; V04.03.01.00	24.01.2018	Denk		bMsg1022, IN_IG.tPB2MM.bParaSetupOk added
; V04.07.00.00	23.01.2019	Zengerer	Distribute Para task with perm messaage handling capability to all modules, no functional change to V4.06
; V04.07.00.00	01.02.2019	Hohensinner	Ignition Information for custom module (bus applications)
; V04.09.00.00	10.12.2019	Denk		Ignition System Self-Test Improvements
; V04.11.00.00	22.12.2021	Andre		Use Para.bSA_Ign_Active to select ignition by SAFI or by MIC
; V04.12.00.00	08.09.2022	Andre		Select the engine speed from the ICxx module also if SEMIC is active
; V04.13.00.00	17.10.2023	Andre		Bugfix for M_STRDRE
;				05-12-2023	Bacci		Added ventilation demand and release before starting the self-test (2023-190)
;				05.03.2024	Bacci		Changes on trip 1061 added
; V04.14.00.00	27.11.2024	Andre		Display B3226 and prevent B3225 during purge starts with all cylinders skipped.
;				02.12.2024	Andre		Set ignition feedback from CAN to TRUE in simulation mode
;				13.02.2025	Andre		ZM2_ZEST not set while the early gas valve opening function is active.
;
; Instructions for use:
; --------------------
; make only changes at the version numbers
;
; Outstandings:
; ------------
;
; *******************************************************************************
;
"<META>"
;
; Module ID
"<MODUL>IG</MODUL>"
;
; Module Version (xx.yy.zz.cc)
"<VERSION>04.14.00.00</VERSION>"
;
; Module Basisupdate Version BU (00-99)
"<BASISUPDATE_VERSION>00</BASISUPDATE_VERSION>"
;
; Optional: specify order number for limitated module usage
"<ORDER></ORDER>" ;<!--(optional for restricted customizations; missing statement makes module valid for all orders)-->
;
; Parameter Check <PARAn Name='aAbcdef' MIN='xxx' MAX='yyy' />  (watch for correct spacings and apostrophs!)
"<PARAMETER_CHK>"
"	<PARA1 Name='iEng_Motortype' MIN='208' MAX='920' />"
"	<PARA2 />"
"	<PARA3 />"
"	<PARA4 />"
"	<PARA5 />"
"</PARAMETER_CHK>"
;
; Statement, if engine operation is also allowed without this module (FALSE) or if this module´s parameter check passing is mandatory (TRUE)
"<MANDATORYMODULE>TRUE</MANDATORYMODULE>"
;
; Permanent Datamodule Filenames<!-- enter filenames for counter and INTERNAL parameter only; filename without extention-->
"<DATAMODULES>" ;<!-- optional; mehrere DATAMODULES erlaubt-->
"	<DATAMODULE>par_IG</DATAMODULE>"
"</DATAMODULES>"
;
; Dependencies Modules (MMxx.yy.zz.cc)
"<DEPENDENCIES>"
"	<DEPENDENCY MODULE='SY' VERSION='04.00.00.00' />"
"	<DEPENDENCY MODULE='PB' VERSION='04.00.00.00' />"
"	<DEPENDENCY MODULE='SA' VERSION='04.00.00.00' />"
"	<DEPENDENCY MODULE='OP' VERSION='04.00.00.00' />"
"	<DEPENDENCY MODULE='MO' VERSION='04.00.00.00' />"
"	<DEPENDENCY MODULE='IC' VERSION='04.13.00.00' />"
"	<DEPENDENCY MODULE='HA' VERSION='04.13.00.00' />"
"	<DEPENDENCY MODULE='GT' VERSION='04.00.00.00' />"
"	<DEPENDENCY MODULE='EG' VERSION='04.00.00.00' />"
"	<DEPENDENCY MODULE='EC' VERSION='04.00.00.00' />"
"	<DEPENDENCY MODULE='AG' VERSION='04.14.00.00' />"
"	<DEPENDENCY MODULE='AB' VERSION='04.00.00.00' />"
"	<DEPENDENCY MODULE='GC' VERSION='04.03.00.00' />"
"	<DEPENDENCY MODULE='VE' VERSION='04.13.00.00' />"
"   <DEPENDENCY VISVERSION='02.12.03.00' />"			; Dependencies Visualization
"</DEPENDENCIES>"
;
; Module function description
"<MODULEFUNCTION>" ;<!-- short overview documentation of module function; add reference to detailed information, if available-->
"	<General>	"
"	 Handling of general ignition topics	"
"	</General>	"
""
"	<F1 Name='Engine speed' LastModified='04.00.00.00'>"
"	Engine speed handling depending on used ignition system. 	"
"	</F1>"
"	<F2 Name='Ignition voltage calculations' LastModified='04.00.00.00'>"
"	 Calculation of min, max and avg values depending on used ignition system.	"
"	</F2>"
"	<F3 Name='Timing point calculation' LastModified='04.00.00.00'>"
"	 Calculation of ignition timing point min, max and avg values depending on used ignition system. "
"	</F3>"
"	<F4 Name='Ignition selftest' LastModified='04.00.00.00'>"
"	Ignition system selftest mode functionallity. "
"	</F4>"
"	<F5 Name='Double Ignition' LastModified='04.00.00.00'>"
"	Double ignition functionallity and building of variable bIgn_Run. "
"	</F5>"
""
"	<Info>"
"	V4.01.00	01-07-2014	Denk 	MM2VIS.bIgn_SelfTest added	"
"   V4.01.00	09.07.2014	Denk	OUT_IG.rCA_Ign_Avg := ZZPAvg; added  "
"   V4.05.00	21.12.2017	Denk	Bugfix, ignition self test with IC/MIC	  "
"	</Info>"
""
"	<Customized LastModified='4.0.0.0'>	"
"	- Nothing "
"	</Customized>	"
""
"</MODULEFUNCTION>"
;
"</META>"
```

### Module_IG.typ - Module global data types
```iecst
TYPE
	IN_IG_Struct : 	STRUCT
		tPB2MM : ParaBase2MM_type; (*Data exchange structure to ParaBase*) (*OldName:new PV; Cycle:5;*)
		tAB2IG : AmmBase2MM; (*AMM structure*) (*OldName:new PV; Cycle:2;*)
		tIgn_Run_Hal : HALioDi_Type; (*DI: Ignition system running*) (*OldName:ZIB;Cycle:2;*)
		tIgn2_Run_Hal : HALioDi_Type; (*DI: Ignition system double running*) (*OldName:ZIB2; Cycle:2;*)
		tGCB_RUC : HALioDo_Type; (*DO: Generator circuit breaker release under voltage coil*) (*OldName:A_USP; Cycle:2;*)
		tIgn_OverspeedRelay : HALioDi_Type; (*DI: Overspeed relay *) (*OldName:UEDZ; Cycle:5;*)
		tGCB_On : HALioDi_Type; (*DI: generator circuit breaker closed *) (*OldName:GCB_ON; Cycle:5;*)
		bIgnOperating : BOOL; (*SAFI ignition system running*) (*OldName:ZIB; Cycle:2;*)
		bMsg1026 : BOOL; (*shutdown failure*) (*OldName:M_ANSTAB; Cycle:2;*)
		bIgn_Dem : BOOL; (*demand ignition*) (*OldName:ZUEND; Cycle:2;*)
		bIgn_Dem_TC5 : BOOL; (*demand ignition*) (*OldName:ZUEND; Cycle:2;*)
		bGV_On : BOOL; (*Command open gas valves*) (*OldName:M_GASV; Cycle:2;*)
		bGV_On_TC2 : BOOL; (*Command open gas valves*) (*OldName:M_GASV; Cycle:2;*)
		rCA_IgnP_Set : REAL; (*global ignition timing set point*) (*OldName:W_ZZP ; Cycle:2;*)
		rCA_Ign_Act : ARRAY[0..24]OF REAL; (*actual ignition timing *) (*OldName:ActTiming; Cycle:2;*)
		rN_IgnIC_Act : REAL; (*engine speed meassured by ignition *) (*OldName:ZDGSpeed; Cycle:2;*)
		rN_IgnSAFI_Act : REAL; (* engine speed meassured by ignition *) (*OldName:ZDGSpeed; Cycle:2;*)
		bPr_EOP_Prelub1 : BOOL; (* Vorschmierdruck 1 Pumpe *) (*OldName:AN_VSD1; Cycle:5;*)
		b_IgnIC_SelfTestBack : BOOL; (* switch ignition system to selftest *) (*OldName:GoSelftest; Cycle:5;*)
		b_IgnSAFI_SelfTestBack : BOOL; (* switch ignition system to selftest *) (*OldName:GoSelftest; Cycle:5;*)
		rU_IgnSAFI_Cyl : ARRAY[0..24]OF REAL; (*ignition voltage for each cylinder SAFI*) (*OldName:V_Zyl; Cycle:2;*)
		rU_IgnMon_Cyl : ARRAY[0..24]OF REAL; (*ignition voltage for each cylinder Monic*) (*OldName:V_Zyl; Cycle:2;*)
		bEng_Dem : BOOL; (*module demanded*) (*OldName:M_AGFD; Cycle:2;*)
		bDeflagrationPrct : BOOL; (*Deflagration protection*) (*OldName:PUFF; Cycle:2;*)
		bMnsOk : BOOL; (*Mains ok *) (*OldName:NE_OK; Cycle:5;*)
		bPr_EOP_Prelub2 : BOOL; (*Prelubrication pressure 2 pumps*) (*OldName:AN_VSD2; Cycle:5;*)
		bRelEngTurn_OilSkid : BOOL; (*release engine barring gear (Durchdrehvorrichtung) from Oil Skid*) (*OldName:new pv;Cycle:5*)
		bEngOilLevel_Lo : BOOL; (* engine oil level low *) (*OldName:ZM_OMIN; Cycle:5*)
		tSafetyLoop_EmStop : HALioDi_Type; (*safety loop - emergency stop*) (*OldName: DI_SIS; Cycle: 5;*)
		tSafetyLoop_Eng : HALioDi_Type; (*safety loop - engine*) (*OldName: RUHE, DI_RUHE_TC1; Cycle: 5;*)
		bSimWinMOD_Active : BOOL; (*WinMode simulation active *) (* OldName:new PV; Cycle:5*)
		iIdx_OMSS : INT; (* inex of operation mode selector switch - 0..OFF, 1..MAN, 2..AUTO, 3..TEST, 4..SCAVENGING *) (*OldName:new PV;Cycle:5;*)
		bInLouRelVE : BOOL; (*inlet louvers open or not closed*)
		bIC_Ign_Run_CAN : BOOL; (*IC Output ignition active from CAN*)
		bTOF_HwBypassDigitalTwin : BOOL; (*Hardware bypass digital twin - T3 adaptive cranking time*)
		bMsg2295 : BOOL; (*engine room ventilation failure inlet air*)
		bMissfCyl_PurgeCrk : BOOL; (*skip fire all cylinders while purging*)
	END_STRUCT;
	OUT_IG_Struct : 	STRUCT
		tIG2PB : MM2ParaBase_type; (*Data exchange structure to ParaBase*) (*OldName:new PV; Cycle:5;*)
		tIG2AB : MM2AmmBase; (*AMM structure*) (*OldName:new PV; Cycle:5;*)
		rN_EngAct : REAL; (*Engine Speed (1/min)*) (*OldName:ZDGSpeed; Cycle:2;*)
		bEO_PrelubeDemIgn : BOOL; (*Demand Prelubricating from ignition*) (*OldName:PRELUBE_IgnST; Cycle:2;*)
		bIgn_SelfTest : BOOL; (*Switch ignition system to selftest *) (*OldName:GoSelftest; Cycle:5;*)
		b_ST_DemIgn : BOOL; (*Demand starter from ignition*) (*OldName:STARTER_IgnST; Cycle:5;*)
		rU_Ign_Cyl : ARRAY[0..24]OF REAL; (*Ignition voltage for each cylinder *) (*OldName:V_Zyl; Cycle:;*)
		rU_Ign_Max : REAL; (* Maximum Ignition voltage *) (*OldName:AvgVolt; Cycle:;*)
		bIgn_Run : BOOL; (*Ignition system is running*) (*OldName:ZIB; Cycle:2;*)
		bN_EngStartDrop : BOOL; (*Engine start-up speed drop down*) (*OldName:M_STRDRE; Cycle:2;*)
		bMsg1022 : BOOL; (*Message*) (*OldName:M_UEDZ; Cycle:5;*)
		bIgn2_Sel : BOOL; (*TRUE = Double ignition selected*) (*OldName:IIXZUEND; Cycle:2;*)
		bMsg1064 : BOOL; (*Message *) (*OldName:M_UEDZRP; Cycle:5;*)
		bMsg3561 : BOOL; (*	Message	*) (*OldName:bPv; Cycle:5;*)
		tCA_IgnP_Set : HALioAo_Type; (*AO: timing point*) (*OldName:ssZZPOutWE; Cycle:2;*)
		bSelfTestRunning : BOOL;
		rCA_Ign_Avg : REAL; (*Actual ignition point average*) (*OldName:ZZPAvg; Cycle:;*)
		rU_Ign_Avg : REAL; (* *) (*OldName:AvgVolt; Cycle:;*)
		rU_Ign_Min : REAL; (* *) (*OldName:MinVolt; Cycle:;*)
		rCA_Ign_Min : REAL; (*Actual min. cylinder ignition point*) (*OldName:ZZPMin; Cycle:;*)
		rCA_Ign_Max : REAL; (*Actual max. cylinder ignition point*) (*OldName:ZZPMax; Cycle:;*)
		iIdx_IgnSelfTest : INT; (*Number of shown picture regarding step of execution. 0 - 50 in steps of 10. Detailded description in every step where used.*) (*OldName:usP5xSelftestStep; Cycle:;*)
		bInLouDemIgn : BOOL; (*Inlet louver demand for ignition selftest*)
		bIgn_Run_CAN : BOOL; (*Ignition system is running - feedback from CAN*)
	END_STRUCT;
	Para_IG_Struct : 	STRUCT
		bIgnMon_Active : BOOL; (*PARA [12064]: TRUE = MONIC is enabled/active*) (*OldName:monic_vis; Cycle:;*)
		bSA_Active : BOOL; (*PARA [12114]: TRUE = SAFI is enabled/active*) (*OldName:bSA_Active; Cycle:;*)
		b_IgnIC_900Active : BOOL; (*PARA [12062]: TRUE = CAN ignition system is used *) (*OldName:ic900_vis; Cycle:;*)
		bSA_Ign_Active : BOOL; (*PARA [12117]: TRUE = SAFI ignition function is enabled/active*) (*OldName:bSAFIIgn_Act; Cycle:;*)
		bIgn2_Sel_Para : BOOL; (*PARA [12063]: Select double ignition*) (*OldName:sel_2ignition; Cycle:;*)
		rN_EngStart_HyHi : REAL; (*PARA [11295]: speed engine start limit high hysteresis*) (*OldName:HY_DREHZ; Cycle:;*)
		rN_EngStart_LimHi : REAL; (*PARA [11296]: speed engine start limit high*) (*OldName:GW_DREHZ; Cycle:;*)
		rN_EngStartMon_HyHi : REAL; (*PARA [12067]: speed engine start monitoring limit high hysteresis*) (*OldName:HY_STRDRE; Cycle:;*)
		rN_EngStartMon_LimHi : REAL; (*PARA [12068]: speed engine start monitoring limit high*) (*OldName:GW_STRDRE; Cycle:;*)
		iEng_Motortype : INT; (*PARA: Motortype of the engine*) (*OldName:motortyp; Cycle:;*)
		rCA_RetTimeLim : REAL; (*PARA [12066]: Retard ignition timing limit*) (*OldName:RetTimLi; Cycle:;*)
		rCA_AdvTimeLim : REAL; (*PARA [12065]: Advanced ignition timing limit*) (*OldName:AdvTimLi; Cycle:;*)
		rN_PLC_LimHi : REAL; (*PARA [12070]: Overspeed PLC limit *) (*OldName:GW_UEDZ; Cycle:;*)
		rN_PLC_HyHi : REAL; (*PARA [12069]: Overspeed PLC hysteresis *) (*OldName:HY_UEDZ; Cycle:;*)
		tiIgn_SelfTest : TIME; (*PARA [14432]: Ignition self test duration*) (*OldName:monic_vis; Cycle:;*)
		bSEMIC_Active : BOOL; (*PARA[14519]: Ignition controller SEMIC*)
	END_STRUCT;
	MM2VIS_Struct : 	STRUCT
		rCA_Ign_Act : ARRAY[0..24]OF REAL; (*actual cylinder ignition point*) (*OldName:ActTiming; Cycle:;*)
		rCA_Ign_Avg : REAL; (*Actual ignition point average*) (*OldName:ZZPAvg; Cycle:;*)
		rCA_Ign_Min : REAL; (*Actual min. cylinder ignition point*) (*OldName:ZZPMin; Cycle:;*)
		rCA_Ign_Max : REAL; (*Actual max. cylinder ignition point*) (*OldName:ZZPMax; Cycle:;*)
		iIdx_IgnSelfTest : INT; (*Number of shown picture regarding step of execution. 0 - 50 in steps of 10. Detailded description in every step where used.*) (*OldName:usP5xSelftestStep; Cycle:;*)
		rU_Ign_Cyl : ARRAY[0..24]OF REAL; (*ignition voltage for each cylinder *) (*OldName:V_Zyl; Cycle:;*)
		rU_Ign_Avg : REAL; (* *) (*OldName:AvgVolt; Cycle:;*)
		rU_Ign_Max : REAL; (* *) (*OldName:MaxVolt; Cycle:;*)
		rU_Ign_Min : REAL; (* *) (*OldName:MinVolt; Cycle:;*)
		bMsg3346 : BOOL; (* *) (*OldName:; Cycle:;*)
		bMsg3228 : BOOL; (* *) (*OldName:; Cycle:;*)
		bMsg3347 : BOOL; (* *) (*OldName:; Cycle:;*)
		bMsg1061 : BOOL; (* *) (*OldName:; Cycle:;*)
		bMsg3225 : BOOL; (* *) (*OldName:; Cycle:;*)
		bMsg3226 : BOOL; (* *) (*OldName:; Cycle:;*)
		bMsg1022 : BOOL; (* *) (*OldName:; Cycle:;*)
		bMsg1064 : BOOL; (* *) (*OldName:; Cycle:;*)
		bMsg3561 : BOOL; (* *) (*OldName:; Cycle:;*)
		rN_EngAct : REAL; (*Engine Speed (1/min)*) (*OldName:; Cycle:;*)
		bIgn_SelfTest : BOOL; (*Switch ignition system to selftest *) (*OldName:GoSelftest; Cycle:5;*)
		bMsg9044 : BOOL; (* *) (*OldName:; Cycle:;*)
	END_STRUCT;
	VIS2MM_Struct : 	STRUCT
		bIgn_SelfTestStart : BOOL; (*start self test button*) (*OldName:; Cycle:;*)
		bIgn_SelfTestStop : BOOL; (*stop self test button*) (*OldName:; Cycle:;*)
		bIgn_SelfTestPrep : BOOL; (*start preperation button*) (*OldName:; Cycle:;*)
		bIgn_SelfTestCancel : BOOL; (*cancel preperation button*) (*OldName:; Cycle:;*)
		bHVMaxValueAct : BOOL; (*Spark voltage maximum*) (*OldName:; Cycle:;*)
	END_STRUCT;
END_TYPE
```

### Module_IG.var - Module global variables
```iecst
VAR
	M_DREHZ : BOOL; (* Startdrehzahl *)
	AN_STRDRE : BOOL; (* Startdrehzahl *)
	bGnlTrip1_IG : BOOL;
	bGnlTrip2_IG : BOOL;
	bGnlTrip3_IG : BOOL;
	bGnlTrip_IG : BOOL;
	bGnlWarning_IG : BOOL;
	bMsg1061_Set : BOOL; (*Module global variable to set message 1061*)
	iIdx_IgnSelfTest : INT; (*Number of shown picture regarding step of execution. 0 - 50 in steps of 10. Detailded description in every step where used.*)
	IN_IG : IN_IG_Struct;
	MM2VIS : MM2VIS_Struct;
	M_STRDRE : BOOL; (*Engine speed fallen below starter speed *)
	OUT_IG : OUT_IG_Struct;
	Para : Para_IG_Struct;
	ParaFactoryDefault : Para_IG_Struct := (0);
	pm : Para_IG_Struct;
	rU_Ign_Avg : REAL; (*Average ignition voltage*)
	rU_Ign_Max : REAL; (*Maximum ignition voltage*)
	rU_Ign_Min : REAL; (*Minimum ignition voltage*)
	usP5xSelftestStep : UINT;
	VIS2MM : VIS2MM_Struct;
	xEngtype : EngType; (*FB for Engine type specific values*)
	ZEST_1 : BOOL := 0; (*Ignition 1 failure*)
	ZEST_2 : BOOL := 0; (*Ignition 2 failure*)
	ZM1_ZEST : BOOL; (*Ignition failure*)
	ZM2_ZEST : BOOL; (*Ignition failure*)
	ZZPAvg : REAL; (* actual ignition point average *)
	ZZPMax : REAL; (* actual max.cylinder ignition point *)
	ZZPMin : REAL; (* actual min.cylinder ignition point *)
	bNoInitDetected : BOOL := FALSE; (*allways true, except 1cycle on init up*)
END_VAR
```

### Program Logical/Ignition/IGGen (IEC, version 4.14.0) - + General task

- IgnGenCyclic.st (not readable text: treated as protected, skipped)

- IgnGenInit.st (not readable text: treated as protected, skipped)

#### IgnGen.var - Local variables
```iecst
VAR
	ucCylinderCount : USINT;
	rU_IgnSAFI_Cyl : ARRAY[0..24] OF REAL; (*ignition voltage SAFI system for each cylinder local variable*)
	rU_IgnMon_Cyl : ARRAY[0..24] OF REAL; (*ignition voltage IC system for each cylinder local variable*)
	xGR_MAXR_EngSpeed : GR_MAXR; (*Limit max for Engine speed*)
	xGR_MAXR_EngineStartSpeed : GR_MAXR;
	ucCylIndex : USINT;
	rU_Ign_Avg_Sum : REAL; (*Average ignition voltage Temporary*)
	TON_SecondTick1 : TON; (* CAN BUS FAHLER *)
	TON_SecondTick : TON; (* CAN BUS FAHLER *)
	rU_Ign_Calc : ARRAY[0..24] OF REAL; (*ignition for each cylinder local variable*)
	rZZPAvg : REAL;
	bIgn_SelfTest : BOOL;
END_VAR
```

### Program Logical/Ignition/2xzuend (IEC, version 4.11.0) - + Double ignition

- 2xzuendCyclic.st (not readable text: treated as protected, skipped)

- 2xzuendInit.st (not readable text: treated as protected, skipped)

#### 2xzuend.var - Local variables
```iecst
VAR
	xTONIgn1FaultDelay : TON; (*Ignition1 fault delay *)
	xTONIgn2FaultDelay : TON; (*Ignition 2 fault delay *)
END_VAR
```

### Program Logical/Ignition/Selftest (IEC, version 4.13.0) - + Ignition selftest

- Selftest.st (not readable text: treated as protected, skipped)

#### Selftest.typ
```iecst
TYPE
	trafficLight_typ : 	STRUCT
		usP5xLightRed : UINT; (*Color of the traffic light*)
		usP5xLightYellow : UINT; (*Color of the traffic light*)
		usP5xLightGreen : UINT; (*Color of the traffic light*)
	END_STRUCT;
	Cylinder : 	STRUCT
		Selection : UINT;
		Data : ARRAY[0..24]OF UINT;
		Cyl : ARRAY[0..24]OF CylVal;
	END_STRUCT;
	CylVal : 	STRUCT
		Exh_Temp : INT;
		Spark_IP : INT;
		Spark_HV : INT;
		Knock_Int : INT;
		Knock_mV : INT;
		Valve_mV : INT;
		Press_bar : INT;
	END_STRUCT;
	bargraphScal_typ : 	STRUCT
		scScalEndValue : ARRAY[0..1]OF SINT; (*Start of the right limit area*)
		scScalStartValue : ARRAY[0..1]OF SINT; (*End of the left limit area*)
		scScalMaxDatapoint : ARRAY[0..1]OF SINT; (*Maximum value of the scale area*)
		scScalMinDatapoint : ARRAY[0..1]OF SINT; (*Minimum value of the scale area*)
		scBarValue : SINT; (*Value of the bargraph*)
		tShowBar : showBarColor_typ; (*Structur to show the OK-Bar (green) or the ERROR-Bar (red)*)
	END_STRUCT;
	showBarColor_typ : 	STRUCT
		ucStatusBarAct : USINT; (* Statusdatapoint for the GREEN Avg. Bar *)
		ucStatusBarMax : USINT; (* Statusdatapoint for the RED Limit Max Bar *)
		ucStatusBarMin : USINT; (* Statusdatapoint for the BLUE Limit Min Bar *)
	END_STRUCT;
	bargraphLeftRight_typ : 	STRUCT
		ucBarLeft : USINT; (*Value of the left bargraph*)
		ucBarRight : USINT; (*Value of the right bargraph*)
		scLimitLeft : SINT; (* Limitvalue to the left side *)
		scLimitRight : SINT; (* Limitvalue to the right side *)
		tShowBar : showBarLeftRight_typ; (*Structur to show the OK-Bar (green) or the ERROR-Bar (red)*)
	END_STRUCT;
	showBarLeftRight_typ : 	STRUCT
		ucStatusBarLeftAct : USINT; (* Statusdatapoint for the GREEN Avg. Bar *)
		ucStatusBarRightAct : USINT; (* Statusdatapoint for the GREEN Avg. Bar *)
		ucStatusBarMax : USINT; (* Statusdatapoint for the RED Limit Max Bar *)
		ucStatusBarMin : USINT; (* Statusdatapoint for the BLUE Limit Min Bar *)
	END_STRUCT;
END_TYPE
```

#### Selftest.var
```iecst
VAR
	xTON_SelftestPrelubCancel : TON;
	xTON_SelftestStarterWait : TON;
	xTON_SelftestStarter : TON;
	xTON_SelftestWait : TON;
	xTON_SelftestText : TON;
	bIgn_SelfTestBack : BOOL; (* switch ignition system to selftest, feedback ON signal from ignition systems*)
	xTON_SelftestBack : TON;
	tiSelftestBack : TIME := T#2s;
	xTON_SelfTest_Duration : TON;
END_VAR
```

### Program Logical/Ignition/MsgIG (IEC, version 4.14.0) - + Messages

- MsgIGCyclic.st (not readable text: treated as protected, skipped)

- MsgIGInit.st (not readable text: treated as protected, skipped)

#### MsgIG.var - Local variables
```iecst
VAR
	GR_MAX_OvrSpd : GR_MAXR;
	xMsg3561 : Msg;
	iAdrAmmBase2MM : UDINT;
	iAdrMM2AmmBase : UDINT;
	xMsg1061 : Msg;
	xMsg1022 : Msg;
	xMsg1064 : Msg;
	xMsg3225 : Msg;
	xMsg3226 : Msg;
	xMsg3228 : Msg;
	xMsg3346 : Msg;
	xMsg3347 : Msg;
	TP_R_GridOK : TP_R;
	bOverspdPLC : BOOL;
	T76 : BOOL; (*Ignition failure*)
	xTONIgnFail : TON; (*Ignition failure *)
	xTON_OpenGV_Mon : TON;
	xMsg9044 : Msg;
	SR_M_STRDRE : SR;
END_VAR
```

### Program Logical/Ignition/VisIG (IEC, version 4.01.0) - + Visualization task

- VisIGCyclic.st (not readable text: treated as protected, skipped)

- VisIGInit.st (not readable text: treated as protected, skipped)

### Program Logical/Ignition/ParIG (IEC, version 4.06.0) - + Parameter handling

- perm_par.st (not readable text: treated as protected, skipped)

#### perm_par.var
```iecst
VAR
	tParaIntern : ParaHandler_typ; (*Connector type to perm_par*)
	tMM2ParaBase_ReadBack : MM2ParaBase_type; (*INTERNAL! V4.06 new readback structure for information from previous tasks*)
	bWriteDataObj : BOOL; (* TRUE=write data object module *)
	bDataObjLenErr : BOOL; (*Error occured in permem: data module size missmatch*)
	bCreateDataObj : BOOL; (* TRUE=create new data object *)
	bWriteOnce : BOOL; (* write permanent memory once *)
	DatObjCreate_01 : DatObjCreate; (* data object create *)
	DatObjInfoBak_02 : DatObjInfo; (* data object info *)
	DatObjDelete_01 : DatObjDelete; (* data object delete *)
	DatObjRead_01 : DatObjRead; (* data object read *)
	DatObjRead_02 : DatObjRead; (* manual initiated data object read *)
	DatObjWrite_01 : DatObjWrite; (* data object write *)
	DatObjDelete_02 : DatObjDelete; (* data object delete *)
	DatObjDelete_11 : DatObjDelete; (*Delete Backup File*)
	DatObjInfo_01 : DatObjInfo; (* data object info *)
	DatObjInfo_02 : DatObjInfo; (* data object info *)
	szModuleName : STRING[35]; (* module name of object *)
	szModuleNameBackup : STRING[35]; (* module name of posiibly created backup object *)
	DatObjCopy_01 : DatObjCopy;
	bCopyDataObj : BOOL;
	TON_WarnDelay : TON;
	TON_WritePMEM : TON; (* delay write permanent memory *)
	ulPMPointer : UDINT; (* adress of actual checksum value *)
	ulChecksum : UDINT; (* parameter checksum value *)
	pm_len : UDINT; (* permanent value lenght *)
	ulChecksumOld : UDINT; (* last vlaue of parameter checksum *)
	ulChkValue : UDINT; (* actual value of parameter pointer *)
	pm_id : UDINT; (* permanent value identifier *)
	pm_p : UDINT; (* permanent value pointer *)
	DatObjInfo_META : DatObjInfo;
	DatObjRead_META : DatObjRead;
	szMetaDataRaw : STRING[2000];
	szMetaData : ARRAY[0..4] OF STRING[35];
	szMetaDataVis : ARRAY[0..3] OF STRING[35];
	ssIndex : INT;
	ssCount : INT;
	ucMetaDataRaw : ARRAY[0..2000] OF USINT;
	ssCount2 : INT;
	szMetaDataFile : STRING[10];
	szText1 : STRING[20];
	pv_adr_IN_XX_tPB2MM : UDINT;
	pv_lng : UDINT;
	pv_lng_IN_XX_tPB2MM : UDINT;
	pv_lng_OUT_XX_tPB2MM : UDINT;
	szText2 : STRING[20];
	pv_adr_OUT_XX_tXX2PB : UDINT;
END_VAR
VAR CONSTANT
	ERR_NOERROR : UINT := 0;
END_VAR
VAR
	usPMWriteCnt : UINT;
	pm_Error : UDINT; (* permanent value error *) (* Deleted: pm : ParaMem_typ; permanent memory tags mathias, 22.8.11*)
	fun_Error : UDINT := 0; (*state > 0 = function error*)
	xLocalParaCheck : ParaCheckFUB; (*local function instance to check parameter values*)
	TON_ParaSetupOk : TON;
	bParaCheckSystemOk : BOOL;
	iDebug_ParaOkChecked : UDINT;
	bRestoreBackupDataObj : BOOL := FALSE;
	bRestoreDataObjContent : BOOL := FALSE;
	pm_id_backup : UDINT;
	pm_p_Backup : UDINT;
	DatObjCopy_02 : DatObjCopy;
	bDeleteBackupDataObj : BOOL := FALSE; (*Command to delete backup data module file on purpose*)
	bDebugPara : ARRAY[0..5] OF BOOL;
	ssIndex2 : INT;
	ssIndex3 : INT;
	ssIndex4 : INT;
	ssIndexVis : INT;
	szText : STRING[40];
	pv_adr_Para : UDINT;
	szParaSnippet : ARRAY[0..5] OF STRING[150];
	szParaIndex : STRING[10];
	slValue : DINT;
	iModuleDLD_ResetCount : INT;
	bDownloadDetected : BOOL;
	bFlagParaStructCopyWorking : BOOL; (*true, if cyclic para copying is active, 1 false cycle at every copy *)
	bStoreInitParaInDataObj : BOOL := FALSE;
	bTestflag : BOOL;
	bReadOutMETA_Once : BOOL;
	tParaCheck_iPvAdress : ARRAY[0..5] OF UDINT;
	tParaCheck_iPvLengt : ARRAY[0..5] OF UDINT;
	tParaCheck_rPvValue : ARRAY[0..5] OF REAL;
	tParaCheck_rRangeMIN : ARRAY[0..5] OF REAL;
	tParaCheck_rRangeMAX : ARRAY[0..5] OF REAL;
	tParaCheck_szPvName : ARRAY[0..5] OF STRING[35];
	ssFormatDetected : INT;
	szMetaDataPart : STRING[150];
	szFullTaskName : STRING[35];
	szFullMetaModuleName : STRING[35];
	debugLen : INT;
	debugSize : INT := 0;
	strcat_adr1 : UDINT;
	strcat_adr2 : UDINT;
	ssIndexTN : INT;
	bAlternate : BOOL;
	n : INT;
	iAlternateChecksum : DINT;
	iAlternateChecksumOld : DINT;
	ulDebugChkValue : ARRAY[0..999] OF UDINT;
	Adr1 : UDINT;
	Adr2 : UDINT;
	usPMWriteCntStepsize : UINT := 1; (*different step sizes to help debug*)
	usPMWriteCntXOR : UINT;
	usPMWriteCntAltSum : UINT;
	ulAdrPM : UDINT;
	usChkValuePM : USINT;
	ulAdrPara : UDINT;
	ulPara_len : UDINT;
	usChkValuePara : USINT;
	iDebugCountPMDifferences : DINT := 0;
	bEngineRunDetected : BOOL; (*detection status bit autocommand 100 /101  for engine run state*)
	ucMetaDataDebugInfoLine : ARRAY[0..24] OF STRING[80];
	ssIndexMand : INT := 0;
	szMetaDataMand : STRING[35];
	iMyErrorInfo_Autoreset : DINT; (*internal autoreset counter*)
	ssIndex_Version : INT; (*internal*)
	ssIndex_BU : INT; (*internal*)
	ssIndex_BU2 : INT; (*internal*)
END_VAR
```

### Package Logical/KLS98 - KL: KLS98

### Data object Logical/KLS98/META_KL (Simple) - Simple data object.

#### META_KL.dat
```
; *******************************************************************************
; AGGR: Module Meta Data (data module)
;
; This code is confidential and proprietary to the INNIO Company.
; It may not be used in any form, or reproduced in any manner, without the express
; written permission of the INNIO Company.
; Copyright, INNIO Company, 2019
;
; Customized modifications: -
; ------------------------
;
; History:
; -------
; V3.99		06-03-2013	Weitzer, generated for modular software
; V4.00 	11-09-2013      pankajrodey, updated file with relevant information
; V4.00 	31.01.2014	Weitzer, versions changed
; V4.01 	15-07-2014	Weitzer, add CAN communication tasks
; V4.02		02-06-2015	Caks, added two OUT interfaces
; V4.04 	20-03-2017	Perktold, version changed
; V4.04		15.05.2017	Gwiggner, KLS98 validation - MSF not working
; V4.05		27.07.2017	Messner, CAN Diagnosis Picture added
; V4.05.01 	16.04.2018	Perktold,	Integrated comments regarding "Safety-related application software source code (EN 13849-1 / 4.6.3)"
;
; Instructions for use:
; --------------------
; make only changes at the version numbers
;
; Outstandings:
; ------------
;
; *******************************************************************************
;
"<META>"
;
; Module ID
"<MODUL>KL</MODUL>"
;
; Module Version (xx.yy.zz.cc)
"<VERSION>04.06.00.00</VERSION>"
;
; Basisupdate Module Version (BU)
"<BASISUPDATE_VERSION>00</BASISUPDATE_VERSION>"
;
; Optional: specify order number for limitated module usage
"<ORDER></ORDER>" ;<!--(optional for restricted customizations; missing statement makes module valid for all orders)-->
;
; Parameter Check <PARAn Name='aAbcdef' MIN='xxx' MAX='yyy' />  (watch for correct spacings and apostrophs!)
"<PARAMETER_CHK>"
"	<PARA1 Name='iEng_Motortype' MIN='208' MAX='920' />"
"	<PARA2 Name='rKLS98_PosResImp' MIN='-720' MAX='720' />"
"	<PARA3 />"
"	<PARA4 />"
"	<PARA5 />"
"</PARAMETER_CHK>"
;
; Permanent Datamodule Filenames<!-- NAME ist ohne Dateiendung einzutragen; Nur für Counter und interne Parameter verwenden-->
"<DATAMODULES>" ;<!-- optional; mehrere DATAMODULES erlaubt-->
"	<DATAMODULE>par_KL</DATAMODULE>"
"</DATAMODULES>"
;
; Dependencies Modules (MMxx.yy.zz.cc)
"<DEPENDENCIES>"
"	<DEPENDENCY MODULE='AB' VERSION='04.00.00.00' />"
"	<DEPENDENCY MODULE='PB' VERSION='04.00.00.00' />"
"	<DEPENDENCY MODULE='OP' VERSION='04.00.00.00' />"
"	<DEPENDENCY MODULE='IG' VERSION='04.00.00.00' />"
"	<DEPENDENCY MODULE='HA' VERSION='04.00.00.00' />"
"   <DEPENDENCY VISVERSION='02.01.00.00' />"			; Dependencies Visualization
"</DEPENDENCIES>"
;
; Module function description
"<MODULEFUNCTION>" ;<!-- short overview documentation of module function; add reference to detailed information, if available-->
"	<General>	"
"	KLS98 device is equipped with knock sensors for 2 cylinders. The KLS98 module performs the real-time pre-processing of cylinder pressure signals "
"	</General>	"
""
"	<F1 Name='CAN communication' LastModified='4.0.0.0'>"
"	Manage CAN communication between the KLS98 device and the controller.	"
"	</F1>"
"	<F2 Name='Handling of errors and alarms' LastModified='4.0.0.0'>"
"	The module receives various errors from the KLS98 module over CAN and sends the alarms over OPC to the controller.	"
"	</F2>"
"	<F3 Name='Configuration and parameterization of KLS98' LastModified='4.0.0.0'>"
"	This module sends parameters to the KLS98 device over CAN bus.	"
"	</F3>"
""
"	<Info>"
"	Please enter additional module info here.	"
" 	Update 2014-07-17: rKLS98_PosResImp changed MIN=-720 "
"   V4.04  KLS98 validation - MSF not working "
"   V4.06  Bugfix negative Limit + spacer in META_KL"
"	</Info>"
""
"	<Customized LastModified='4.0.0.0'>	"
"	- Nothing "
"	</Customized>	"
""
"</MODULEFUNCTION>"
;
"</META>"
```

### module_KLS.typ - Package data types
```iecst
(********************************************************************
 * COPYRIGHT -- INNIO Company
 ********************************************************************
 * Package: Heating_Cooling_Pkg
 * File: module_Heat_Cool.typ
 * Author: 320003156
 * Created: July 06, 2011
 ********************************************************************
 * Data types of package Heating_Cooling_Pkg
 ********************************************************************)

TYPE
	CanDeviceGo : 	STRUCT
		CANDevGo : ARRAY[0..1]OF USINT;
		ECANDevGo : USINT;
	END_STRUCT;
	IN_KLS_Struct : 	STRUCT
		tAB2KL : AmmBase2MM; (* *) (*OldName:new; Cycle: 5*)
		tPB2MM : ParaBase2MM_type; (* *) (*OldName:FGDRPS; Cycle: 5*)
		iIdx_OMSS : INT; (*Operating mode manual*) (*OldName:BWS_HA; Cycle: 5*)
		rN_EngAct : REAL; (*Engine speed 1/min*) (*OldName:n_ist; Cycle: 5*)
		iCANIdent : UDINT; (* CAN identifier from HalIO *) (* OldName:new PV; Cycle:5 *)
		bSimWinMOD_Active : BOOL;
		iECanDevGo : USINT; (* event status CAN device go *) (* OldName:new PV; Cycle:5 *)
		rP_Act_Norm_Filt : REAL; (*actual power related to rP_Nom filtered T=1s*) (*OldName:P_IST; Cycle:5*)
	END_STRUCT;
	OUT_KLS_Struct : 	STRUCT
		rKLS98_X_Window1 : ARRAY[0..24]OF REAL; (* cylinder values of KLS98 window 1 *) (*OldName:Fenst1; Cycle: 5*)
		rKLS98_X_Window2 : ARRAY[0..24]OF REAL; (* cylinder values of KLS98 window 2 *) (*OldName:Fenst2; Cycle: 5*)
		rKLS98_X_Window3 : ARRAY[0..24]OF REAL; (* cylinder values of KLS98 window 3 *) (*OldName:Fenst3; Cycle: 5*)
		rKLS98_X_Window4 : ARRAY[0..24]OF REAL; (* cylinder values of KLS98 window 4 *) (*OldName:Fenst4; Cycle: 5*)
		rKLS98_N_RunningHours : ARRAY[0..24]OF REAL; (* operating hours KLS98 device *) (*OldName:usKLSBetrH; Cycle: 5*)
		rKLS98_Vers_SW : ARRAY[0..24]OF REAL; (*kls98 version*) (*OldName:usKLSVers; Cycle: 5*)
		tKL2AB : MM2AmmBase; (* *) (*OldName:new; Cycle: 5*)
		tKL2PB : MM2ParaBase_type; (* *) (*OldName:new; Cycle: 5*)
		tKLS98_CanGo : CanDeviceGo; (* Start / Stop CAN communication *) (* OldName:CANDevGo; Cycle:5 *)
		bKLS98_Fault : ARRAY[0..24] OF BOOL; (* TRUE= faulty cyl. knocking signal *) (*OldName:bKLS98Fault; Cycle: 5*)
		bKLS98_Signal : ARRAY[0..24] OF BOOL; (* KLS Measurement Signal Knock Sensor *) (*OldName:KLSMS; Cycle: 5*)
		tE_KLS : ARRAY[0..24] OF _tEventKLS; (* CAN events KLS98 *)
		iKLS98CommErrCount : ARRAY[0..24] OF USINT;
	END_STRUCT;
	PARA_KLS_Struct : 	STRUCT
		rKLS98_PosResImp : REAL; (*Position CAMSHAFT Reset*) (*OldName:PosResImp; Cycle: 5*)
		rCA_Win1_B : REAL; (*Window 1 - Start*) (*OldName:WMF1_B; Cycle: 5*)
		rCA_Win1_D : REAL; (*Window 1 - End*) (*OldName:WMF1_D; Cycle: 5*)
		rCA_Win2_B : REAL; (*Window 2 - Start*) (*OldName:WMF2_B; Cycle: 5*)
		rCA_Win2_D : REAL; (*Window 2 - End*) (*OldName:WMF2_D; Cycle: 5*)
		rKLS98_W2_Limit : REAL; (*Window 2 - Limit*) (*OldName:Fenst2LiMn; Cycle: 5*)
		rKLS98_MS_Limit : REAL; (*Measuring Signal failure Fenst2LiMn*) (*OldName:Fenst2LiMx; Cycle: 5*)
		iEng_Motortype : INT; (*Select engine type*) (*OldName:new; Cycle: 5*)
		bKLS98_Active : BOOL; (*Activate KLS*) (*OldName:kls98_vis; Cycle: 5*)
		iKlS_KnckValue_Limit : INT; (*Window 2 - Limit*) (*OldName:Fenst2LiMn; Cycle: 5*)
		iKlS_MSFailure_Limit : INT; (*Measuring Signal failure Fenst2LiMn*) (*OldName:Fenst2LiMx; Cycle: 5*)
	END_STRUCT;
	_tEventKLS : 	STRUCT
		conf : ARRAY[0..99]OF USINT;
	END_STRUCT;
	MM2VIS_Struct : 	STRUCT
		bMsg3131 : BOOL; (*3131*) (*OldName:KLS_CAN[1];Cycle: 5*)
		bMsg3132 : BOOL; (*3132*) (*OldName:KLS_CAN[2];Cycle: 5*)
		bMsg3133 : BOOL; (*3133*) (*OldName:KLS_CAN[3];Cycle: 5*)
		bMsg3134 : BOOL; (*3134*) (*OldName:KLS_CAN[4];Cycle: 5*)
		bMsg3135 : BOOL; (*3135*) (*OldName:KLS_CAN[5];Cycle: 5*)
		bMsg3136 : BOOL; (*3136*) (*OldName:KLS_CAN[6];Cycle: 5*)
		bMsg3137 : BOOL; (*3137*) (*OldName:KLS_CAN[7];Cycle: 5*)
		bMsg3138 : BOOL; (*3138*) (*OldName:KLS_CAN[8];Cycle: 5*)
		bMsg3139 : BOOL; (*3139*) (*OldName:KLS_CAN[9];Cycle: 5*)
		bMsg3140 : BOOL; (*3140*) (*OldName:KLS_CAN[10];Cycle: 5*)
		bMsg3151 : BOOL; (*3151*) (*OldName:KLSSOFTV;Cycle: 5*)
		bMsg3002 : BOOL; (*3002*) (*OldName:KLSFALSOF;Cycle: 5*)
		bMsg3210 : BOOL; (*3210*) (*OldName:KLSZAHN;Cycle: 5*)
		bMsg3211 : BOOL; (*3211*) (*OldName:KLSPAR;Cycle: 5*)
		bMsg3121 : BOOL; (*3121*) (*OldName:KLSCAM[1];Cycle: 5*)
		bMsg3122 : BOOL; (*3122*) (*OldName:KLSCAM[2];Cycle: 5*)
		bMsg3123 : BOOL; (*3123*) (*OldName:KLSCAM[3];Cycle: 5*)
		bMsg3124 : BOOL; (*3124*) (*OldName:KLSCAM[4];Cycle: 5*)
		bMsg3125 : BOOL; (*3125*) (*OldName:KLSCAM[5];Cycle: 5*)
		bMsg3126 : BOOL; (*3126*) (*OldName:KLSCAM[6];Cycle: 5*)
		bMsg3127 : BOOL; (*3127*) (*OldName:KLSCAM[7];Cycle: 5*)
		bMsg3128 : BOOL; (*3128*) (*OldName:KLSCAM[8];Cycle: 5*)
		bMsg3129 : BOOL; (*3129*) (*OldName:KLSCAM[9];Cycle: 5*)
		bMsg3130 : BOOL; (*3130*) (*OldName:KLSCAM[10];Cycle: 5*)
		bMsg3141 : BOOL; (*3141*) (*OldName:KLSTRI[1];Cycle: 5*)
		bMsg3142 : BOOL; (*3142*) (*OldName:KLSTRI[2];Cycle: 5*)
		bMsg3143 : BOOL; (*3143*) (*OldName:KLSTRI[3];Cycle: 5*)
		bMsg3144 : BOOL; (*3144*) (*OldName:KLSTRI[4];Cycle: 5*)
		bMsg3145 : BOOL; (*3145*) (*OldName:KLSTRI[5];Cycle: 5*)
		bMsg3146 : BOOL; (*3146*) (*OldName:KLSTRI[6];Cycle: 5*)
		bMsg3147 : BOOL; (*3147*) (*OldName:KLSTRI[7];Cycle: 5*)
		bMsg3148 : BOOL; (*3148*) (*OldName:KLSTRI[8];Cycle: 5*)
		bMsg3149 : BOOL; (*3149*) (*OldName:KLSTRI[9];Cycle: 5*)
		bMsg3150 : BOOL; (*3150*) (*OldName:KLSTRI[10];Cycle: 5*)
		bMsg3161 : BOOL; (*3161*)
		bMsg3162 : BOOL; (*3162*)
		bMsg3163 : BOOL; (*3163*)
		bMsg3164 : BOOL; (*3164*)
		bMsg3165 : BOOL; (*3165*)
		bMsg3166 : BOOL; (*3166*)
		bMsg3167 : BOOL; (*3167*)
		bMsg3168 : BOOL; (*3168*)
		bMsg3169 : BOOL; (*3169*)
		bMsg3170 : BOOL; (*3170*)
		bMsg3171 : BOOL; (*3171*)
		bMsg3172 : BOOL; (*3172*)
		bMsg3173 : BOOL; (*3173*)
		bMsg3174 : BOOL; (*3174*)
		bMsg3175 : BOOL; (*3175*)
		bMsg3176 : BOOL; (*3176*)
		bMsg3177 : BOOL; (*3177*)
		bMsg3178 : BOOL; (*3178*)
		bMsg3179 : BOOL; (*3179*)
		bMsg3180 : BOOL; (*3180*)
		bMsg3001 : BOOL; (*3001*) (*OldName:KLSSTOER;Cycle: 5*)
		bKLS98_Active : BOOL; (*Activate (*OldName:kls98_vis;Cycle: 5*)
		rKLS98_X_Window2 : ARRAY[0..24]OF REAL; (* cylinder values of KLS98 window 2 *) (*OldName:Fenst2;Cycle: 5*)
		rKLS98_Vers_SW : REAL; (*kls98 version*) (*OldName:usKLSVers; Cycle: 5*)
		iCMSinit_KLS98_status : INT; (* KLS98 Module CMS Init Status *)
		iCMSmain_KLS98_status : INT; (* KLS98 Module Main CMS Status *)
	END_STRUCT;
END_TYPE
```

### module_KLS.var - Package variables
```iecst
(********************************************************************
 * COPYRIGHT -- INNIO Company
 ********************************************************************
 * Package: Heating_Cooling_Pkg
 * File: module_Heat_Cool.var
 * Author: 320003156
 * Created: July 06, 2011
 ********************************************************************
 * Variables of package Heating_Cooling_Pkg
 ********************************************************************)
VAR
	pm : PARA_KLS_Struct;
	Para : PARA_KLS_Struct;
	ParaFactoryDefault : PARA_KLS_Struct := (0);
	OUT_KL : OUT_KLS_Struct := (0);
	IN_KL : IN_KLS_Struct := (0);
	xEngType : EngType := (0);

	kls98_vis : BOOL; (* 1=KLS98 exists *)
	CANopen_error : UINT; (* CAN CONTROLLER STATUS 0=OK *)

	ic900_vis : BOOL; (* TRUE=CAN ignition system is used *)

	ucNumberOfCylinder : USINT; (* number of cylinders *)

	MissfCyl : UDINT; (* cylinder misfire parameter *)
	ZylZahl : USINT; (* number of cylinders for CAN-Comm. *)
	ECANDevGo : USINT; (* event startup parameter CAN device *)
	CANDevGo : ARRAY[0..1] OF USINT; (* startup parameter for CAN devices *)
	KLS98_Node : USINT; (* node number of first KLS98 *)
	KLS98_ID : USINT; (* flag for trigger recipe receive *)
	KLSVers : UINT; (* KLS98 software version number *)
	E_KLS : ARRAY[0..24] OF _tEventKLS;
	ucKLS98CommErrCount : ARRAY[0..24] OF USINT;
	bKLS98Fault : ARRAY[0..24] OF BOOL; (* TRUE= faulty cyl. knocking signal *)
	KLS_CAN : ARRAY[0..10] OF BOOL := [11(0)]; (* KLS CAN KOPPLUNG *)
	usKLSVers : ARRAY[0..24] OF UINT; (*kls98 version*)
	KLS_Err : ARRAY[0..24] OF UINT; (* error status of KLS98 devices *)
	KLSSOFTV : BOOL := 0; (* KLS SOFTWARE VERSIONEN *)
	KLSFALSOF : BOOL := 0; (* KLS FALSCHE SOFTWARE *)
	ucBaureihe : USINT; (* module series *)
	FenstF1 : USINT; (* KLS98 function window 1 *)
	FenstF2 : USINT; (* KLS98 function window 2 *)
	WMF3_B : INT; (* beginn of window 3 in 1/10 deg. *)
	WMF3_D : UINT; (* duration of window 3 in 1/10 deg. *)
	WMF4_B : INT; (* beginn of window 4 in 1/10 deg. *)
	WMF4_D : UINT; (* duration of window 4 in 1/10 deg. *)
	usZahnzahl : UINT; (* number of starter ring gear teeth *)
	PosResImp : INT; (* position reset trigger mark *)
	usFreig_n : UINT; (* speed limit activate KLS functions *)
	ucZuendabst : USINT; (* ignition timing diff. row A to B *)
	FireOrder : ARRAY[0..24] OF USINT; (* engine ignition fire order *)
	KLSGW1 : INT; (* unused KLS98 limit 1 *)
	KLSGW2 : INT; (* unused KLS98 limit 2 *)
	KLSGW3 : INT; (* unused KLS98 limit 3 *)
	KLSGW4 : INT; (* unused KLS98 limit 4 *)
	WMF1_B : INT; (* beginn of window 1 in 1/10 deg. *)
	WMF1_D : INT; (* duration of window 1 in 1/10 deg. *)
	WMF2_B : INT; (* beginn of window 2 in 1/10 deg. *)
	WMF2_D : UINT; (* duration of window 2 in 1/10 deg. *)
	WMF_AB : INT; (* beginn of window misfire in 1/10 *)
	WMF_AD : UINT; (* duration of window misfire in 1/10 *)
	FenstF3 : USINT; (* KLS98 function window 3 *)
	FenstF4 : USINT; (* KLS98 function window 4 *)
	AussSchwel : UINT; (* KLS98 limit for misfire detection *)
	AussInterv : UINT; (* misfire interval cycle parameter *)
	MWFenst1 : INT; (* average parameter for window 1 *)
	MWFenst2 : INT; (* average parameter for window 2 *)
	MWFenst3 : INT; (* average parameter for window 3 *)
	MWFenst4 : INT; (* average parameter for window 4 *)
	Zuendabst : USINT; (* ignition distance from row A to B *)
	StopM : BOOL; (* TRUE=engine is stopped *)
	KLSZAHN : BOOL := 0; (* KLS Falsche Zähnezahl *)
	KLSPAR : BOOL := 0; (* KLS Parameterchecksumfehler *)
	KLSCAM : ARRAY[0..10] OF BOOL := [11(0)]; (* KLS AUSFALL CAM PICKUP *)
	KLSTRI : ARRAY[0..10] OF BOOL := [11(0)]; (* KLS AUSFALL TRIGGER PICKUP *)
	ErrZahnVal : USINT; (* KLS98 with number of teeht error *)
	ErrParVal : USINT; (* KLS98 number with parameter error *)
	Fenst2 : ARRAY[0..24] OF UINT; (* cylinder values of KLS98 window 2 *)
	KLSMS : ARRAY[0..24] OF BOOL := [25(0)]; (* KLS MESSIGNAL KLOPFSENSOR *)
	E_KLS_Err : ARRAY[0..24] OF USINT; (* CAN events KLS98 error messages *)
	KLSSTOER : BOOL := 0; (* KLS Störung *)
	n_ist : INT; (* actual speed [1/min] *)
	LichtMax : ARRAY[0..24] OF UINT; (* cylinder light density from OCA *)
	Fenst1 : ARRAY[0..24] OF UINT; (* cylinder values of KLS98 window 1 *)
	Fenst3 : ARRAY[0..24] OF UINT; (* cylinder values of KLS98 window 3 *)
	Fenst4 : ARRAY[0..24] OF UINT; (* cylinder values of KLS98 window 4 *)
	KLSAktiv : ARRAY[0..24] OF USINT; (* control of active KLS98 functions *)
	Fenst2Max : UINT; (* maximum of values window 2 *)
	Fenst2Min : UINT; (* minimum of values window 2 *)
	KLSVEN : ARRAY[0..24] OF BOOL := [25(0)]; (* KLS Ventilgeräsch maximum *)
	ucFreigabe : ARRAY[0..24] OF USINT; (* control of active KL98 functions *)
	usKLSBetrH : ARRAY[0..24] OF UINT; (* operating hours KLS98 device *)
	E_Fenst1 : ARRAY[0..24] OF USINT; (* CAN event KLS98 window 1 *)
	E_Fenst2 : ARRAY[0..24] OF USINT; (* CAN events KLS98 window 2 *)
	E_Fenst3 : ARRAY[0..24] OF USINT; (* CAN events KLS98 window 3 *)
	E_Fenst4 : ARRAY[0..24] OF USINT; (* CAN events KLS98 window 4 *)
	E_LichtMax : ARRAY[0..24] OF USINT; (* CAN event light maximum *)
	E_Aussetz : ARRAY[0..24] OF USINT; (* CAN events misfire values *)
	bGnlTrip1 : BOOL;
	bGnlTrip2 : BOOL;
	bGnlTrip3 : BOOL;
	bGnlWarning : BOOL;
	bGnlTrip : BOOL;
	BWS_HA : BOOL := 0; (* Betriebswahlschalter Hand/Auto *)
	MM2VIS : MM2VIS_Struct;
	bNoInitDetected : BOOL := FALSE; (*allways true, except 1cycle on init up*)
	CMSmain_KLS98_1 : CMSmain;
	CMSmain_KLS98_2 : CMSmain;
	CMSmain_KLS98_3 : CMSmain;
	CMSmain_KLS98_4 : CMSmain;
	CMSinit_KLS98_x_status : UINT;
	CMSinit_KLS98_1 : CMSinit;
	CMSinit_KLS98_2 : CMSinit;
	CMSinit_KLS98_3 : CMSinit;
	CMSinit_KLS98_4 : CMSinit;
	CMSmain_KLS98_x_status : UINT;
	Aussetz : ARRAY[0..24] OF UINT;
	SIM_rKLS98_X_Window1 : ARRAY[0..24]OF REAL; (* cylinder values of KLS98 window 1 *)
	SIM_rKLS98_X_Window2 : ARRAY[0..24]OF REAL; (* cylinder values of KLS98 window 2 *)
	SIM_rKLS98_X_Window3 : ARRAY[0..24]OF REAL; (* cylinder values of KLS98 window 3 *)
	SIM_rKLS98_X_Window4 : ARRAY[0..24]OF REAL; (* cylinder values of KLS98 window 4 *)
END_VAR
```

### Program Logical/KLS98/EngTypeKL (IEC, version 4.00.0) - + Engine type and firing order selection

- EngTypeKLCyclic.st (not readable text: treated as protected, skipped)

### Program Logical/KLS98/IN_KLS (IEC, version 4.00.0) - + IN variables for KLS98

- IN_KLSCyclic.st (not readable text: treated as protected, skipped)

- Logical/KLS98/kls_98 (protected, skipped)

### Program Logical/KLS98/MsgKLS (IEC, version 4.05.0) - + KLS98 alarms

- MsgKLSCyclic.st (not readable text: treated as protected, skipped)

- MsgKLSInit.st (not readable text: treated as protected, skipped)

#### MsgKLS.var
```iecst
(*******************************************************************************
MsgOL.var

This code is confidential and proprietary to the INNIO Company.
It may not be used in any form, or reproduced in any manner,
without the express written permission of the INNIO Company.
Copyright, INNIO Company, 2019

Customized modifications: -
------------------------

History:
-------
V3.90.0		20-03-2012 pankajrodey 		Created initial structured text code

*******************************************************************************)
VAR
	iAdrAmmBase2MM : UDINT;
	iAdrMM2AmmBase : UDINT;
	xMsg3131 : Msg;
	xMsg3132 : Msg;
	xMsg3133 : Msg;
	xMsg3134 : Msg;
	xMsg3135 : Msg;
	xMsg3136 : Msg;
	xMsg3137 : Msg;
	xMsg3138 : Msg;
	xMsg3139 : Msg;
	xMsg3140 : Msg;
	xMsg3151 : Msg;
	xMsg3002 : Msg;
	xMsg3210 : Msg;
	xMsg3211 : Msg;
	xMsg3121 : Msg;
	xMsg3122 : Msg;
	xMsg3123 : Msg;
	xMsg3124 : Msg;
	xMsg3125 : Msg;
	xMsg3126 : Msg;
	xMsg3127 : Msg;
	xMsg3128 : Msg;
	xMsg3129 : Msg;
	xMsg3130 : Msg;
	xMsg3141 : Msg;
	xMsg3142 : Msg;
	xMsg3143 : Msg;
	xMsg3144 : Msg;
	xMsg3145 : Msg;
	xMsg3146 : Msg;
	xMsg3147 : Msg;
	xMsg3148 : Msg;
	xMsg3149 : Msg;
	xMsg3150 : Msg;
	xMsg3161 : Msg;
	xMsg3162 : Msg;
	xMsg3163 : Msg;
	xMsg3164 : Msg;
	xMsg3165 : Msg;
	xMsg3166 : Msg;
	xMsg3167 : Msg;
	xMsg3168 : Msg;
	xMsg3169 : Msg;
	xMsg3170 : Msg;
	xMsg3171 : Msg;
	xMsg3172 : Msg;
	xMsg3173 : Msg;
	xMsg3174 : Msg;
	xMsg3175 : Msg;
	xMsg3176 : Msg;
	xMsg3177 : Msg;
	xMsg3178 : Msg;
	xMsg3179 : Msg;
	xMsg3180 : Msg;
	xMsg3001 : Msg;
	xMsg3053 : Msg;
	xMsg3054 : Msg;
	xMsg3055 : Msg;
	xMsg3056 : Msg;
	xMsg3057 : Msg;
	xMsg3058 : Msg;
	xMsg3059 : Msg;
	xMsg3060 : Msg;
	xMsg3061 : Msg;
	xMsg3062 : Msg;
	xMsg3063 : Msg;
	xMsg3064 : Msg;
	xMsg3065 : Msg;
	xMsg3066 : Msg;
	xMsg3067 : Msg;
	xMsg3068 : Msg;
	xMsg3069 : Msg;
	xMsg3070 : Msg;
	xMsg3071 : Msg;
	xMsg3072 : Msg;
END_VAR
```

### Program Logical/KLS98/OUT_KLS (IEC, version 4.05.1) - + Out variables for KLS98

- OUT_KLSCyclic.st (not readable text: treated as protected, skipped)

#### OUT_KLS.var - Local variables
```iecst
(********************************************************************
 * COPYRIGHT -- INNIO Company
 ********************************************************************
 * Program: OUT_KLS
 * File: OUT_KLS.var
 * Author: 320003156
 * Created: March 27, 2012
 ********************************************************************
 * Local variables of program OUT_KLS
 ********************************************************************)
VAR
	I : USINT := 0;
	TON_SecondTick : TON;
END_VAR
```

### Program Logical/KLS98/ParKL (IEC, version 4.06.0) - + Parameters KLS98

- perm_par.st (not readable text: treated as protected, skipped)

#### perm_par.var
```iecst
VAR
	tParaIntern : ParaHandler_typ; (*Connector type to perm_par*)
	tMM2ParaBase_ReadBack : MM2ParaBase_type; (*INTERNAL! V4.06 new readback structure for information from previous tasks*)
	bWriteDataObj : BOOL; (* TRUE=write data object module *)
	bDataObjLenErr : BOOL; (*Error occured in permem: data module size missmatch*)
	bCreateDataObj : BOOL; (* TRUE=create new data object *)
	bWriteOnce : BOOL; (* write permanent memory once *)
	DatObjCreate_01 : DatObjCreate; (* data object create *)
	DatObjInfoBak_02 : DatObjInfo; (* data object info *)
	DatObjDelete_01 : DatObjDelete; (* data object delete *)
	DatObjRead_01 : DatObjRead; (* data object read *)
	DatObjRead_02 : DatObjRead; (* manual initiated data object read *)
	DatObjWrite_01 : DatObjWrite; (* data object write *)
	DatObjDelete_02 : DatObjDelete; (* data object delete *)
	DatObjDelete_11 : DatObjDelete; (*Delete Backup File*)
	DatObjInfo_01 : DatObjInfo; (* data object info *)
	DatObjInfo_02 : DatObjInfo; (* data object info *)
	szModuleName : STRING[35]; (* module name of object *)
	szModuleNameBackup : STRING[35]; (* module name of posiibly created backup object *)
	DatObjCopy_01 : DatObjCopy;
	bCopyDataObj : BOOL;
	TON_WarnDelay : TON;
	TON_WritePMEM : TON; (* delay write permanent memory *)
	ulPMPointer : UDINT; (* adress of actual checksum value *)
	ulChecksum : UDINT; (* parameter checksum value *)
	pm_len : UDINT; (* permanent value lenght *)
	ulChecksumOld : UDINT; (* last vlaue of parameter checksum *)
	ulChkValue : UDINT; (* actual value of parameter pointer *)
	pm_id : UDINT; (* permanent value identifier *)
	pm_p : UDINT; (* permanent value pointer *)
	DatObjInfo_META : DatObjInfo;
	DatObjRead_META : DatObjRead;
	szMetaDataRaw : STRING[2000];
	szMetaData : ARRAY[0..4] OF STRING[35];
	szMetaDataVis : ARRAY[0..3] OF STRING[35];
	ssIndex : INT;
	ssCount : INT;
	ucMetaDataRaw : ARRAY[0..2000] OF USINT;
	ssCount2 : INT;
	szMetaDataFile : STRING[10];
	szText1 : STRING[20];
	pv_adr_IN_XX_tPB2MM : UDINT;
	pv_lng : UDINT;
	pv_lng_IN_XX_tPB2MM : UDINT;
	pv_lng_OUT_XX_tPB2MM : UDINT;
	szText2 : STRING[20];
	pv_adr_OUT_XX_tXX2PB : UDINT;
END_VAR
VAR CONSTANT
	ERR_NOERROR : UINT := 0;
END_VAR
VAR
	usPMWriteCnt : UINT;
	pm_Error : UDINT; (* permanent value error *) (* Deleted: pm : ParaMem_typ; permanent memory tags mathias, 22.8.11*)
	fun_Error : UDINT := 0; (*state > 0 = function error*)
	xLocalParaCheck : ParaCheckFUB; (*local function instance to check parameter values*)
	TON_ParaSetupOk : TON;
	bParaCheckSystemOk : BOOL;
	iDebug_ParaOkChecked : UDINT;
	bRestoreBackupDataObj : BOOL := FALSE;
	bRestoreDataObjContent : BOOL := FALSE;
	pm_id_backup : UDINT;
	pm_p_Backup : UDINT;
	DatObjCopy_02 : DatObjCopy;
	bDeleteBackupDataObj : BOOL := FALSE; (*Command to delete backup data module file on purpose*)
	bDebugPara : ARRAY[0..5] OF BOOL;
	ssIndex2 : INT;
	ssIndex3 : INT;
	ssIndex4 : INT;
	ssIndexVis : INT;
	szText : STRING[40];
	pv_adr_Para : UDINT;
	szParaSnippet : ARRAY[0..5] OF STRING[150];
	szParaIndex : STRING[10];
	slValue : DINT;
	iModuleDLD_ResetCount : INT;
	bDownloadDetected : BOOL;
	bFlagParaStructCopyWorking : BOOL; (*true, if cyclic para copying is active, 1 false cycle at every copy *)
	bStoreInitParaInDataObj : BOOL := FALSE;
	bTestflag : BOOL;
	bReadOutMETA_Once : BOOL;
	tParaCheck_iPvAdress : ARRAY[0..5] OF UDINT;
	tParaCheck_iPvLengt : ARRAY[0..5] OF UDINT;
	tParaCheck_rPvValue : ARRAY[0..5] OF REAL;
	tParaCheck_rRangeMIN : ARRAY[0..5] OF REAL;
	tParaCheck_rRangeMAX : ARRAY[0..5] OF REAL;
	tParaCheck_szPvName : ARRAY[0..5] OF STRING[35];
	ssFormatDetected : INT;
	szMetaDataPart : STRING[150];
	szFullTaskName : STRING[35];
	szFullMetaModuleName : STRING[35];
	debugLen : INT;
	debugSize : INT := 0;
	strcat_adr1 : UDINT;
	strcat_adr2 : UDINT;
	ssIndexTN : INT;
	bAlternate : BOOL;
	n : INT;
	iAlternateChecksum : DINT;
	iAlternateChecksumOld : DINT;
	ulDebugChkValue : ARRAY[0..999] OF UDINT;
	Adr1 : UDINT;
	Adr2 : UDINT;
	usPMWriteCntStepsize : UINT := 1; (*different step sizes to help debug*)
	usPMWriteCntXOR : UINT;
	usPMWriteCntAltSum : UINT;
	ulAdrPM : UDINT;
	usChkValuePM : USINT;
	ulAdrPara : UDINT;
	ulPara_len : UDINT;
	usChkValuePara : USINT;
	iDebugCountPMDifferences : DINT := 0;
	bEngineRunDetected : BOOL; (*detection status bit autocommand 100 /101  for engine run state*)
	ucMetaDataDebugInfoLine : ARRAY[0..24] OF STRING[80];
	ssIndexMand : INT := 0;
	szMetaDataMand : STRING[35];
	iMyErrorInfo_Autoreset : DINT; (*internal autoreset counter*)
	ssIndex_Version : INT; (*internal*)
	ssIndex_BU : INT; (*internal*)
	ssIndex_BU2 : INT; (*internal*)
END_VAR
```

### Program Logical/KLS98/VisKL (IEC, version 4.00.0) - + Visu interface for KLS98

- VisKLCyclic.st (not readable text: treated as protected, skipped)

- VisKLInit.st (not readable text: treated as protected, skipped)

#### VisKL.var - Local variables
```iecst
(********************************************************************
 * COPYRIGHT -- INNIO Company
 ********************************************************************
 * Program: VisKL
 * File: VisKL.var
 * Author: 320003156
 * Created: December 11, 2012
 ********************************************************************
 * Local variables of program VisKL
 ********************************************************************)

VAR
iIndex : INT;
END_VAR

VAR CONSTANT

END_VAR
```

- Logical/KLS98/cmskls_1 (protected, skipped)

- Logical/KLS98/cmskls_2 (protected, skipped)

- Logical/KLS98/cmskls_3 (protected, skipped)

- Logical/KLS98/cmskls_4 (protected, skipped)

### Program Logical/KLS98/caniniKL (IEC, version 4.00.0) - + CAN init KLS98

- caniniKLCyclic.st (not readable text: treated as protected, skipped)

### Program Logical/KLS98/canmai (IEC, version 4.00.0) - + CAN main KLS98

- canmaiCyclic.st (not readable text: treated as protected, skipped)

#### canmai.var - Local variables
```iecst
(********************************************************************
 * COPYRIGHT -- INNIO Company
 ********************************************************************
 * Program: canmai
 * File: canmai.var
 * Author: WeitzerT
 * Created: April 15, 2013
 ********************************************************************
 * Local variables of program canmai
 ********************************************************************)
VAR
	ucDeviceSeq : USINT;
END_VAR
```

### Package Logical/Knocking - KN: Knocking Prevention

### Library Logical/Knocking/Lib_KN/lMeNoiAL (ANSIC)

#### lMeNoiAL.fun
```iecst
FUNCTION_BLOCK fMeNoiAL
  VAR_INPUT
    ssMethodType: SINT;
  END_VAR  VAR_INPUT
        Para : tMeNoiAL_PARA; (**)
  END_VAR
  VAR_INPUT
        In : tMeNoiAL_IN; (**)
  END_VAR
 VAR_OUTPUT
        Out : tMeNoiAL_OUT; (**)
  END_VAR
 VAR_OUTPUT
        Dbg : tMeNoiAL_DBG; (**)
  END_VAR
  VAR_OUTPUT
        Version : UDINT; (**)
  END_VAR
	VAR
		bur_BlockIO_MeNoiAL : BlockIO_MeNoiAL;
	END_VAR
	VAR
		bur_D_Work_MeNoiAL : D_Work_MeNoiAL;
	END_VAR
	VAR
		bur_ExternalOutputs_MeNoiAL : ExternalOutputs_MeNoiAL;
	END_VAR
END_FUNCTION_BLOCK
```

#### lMeNoiAL.typ
```iecst
TYPE

   tMeNoiAL_DBG : STRUCT
        uMeNoi_Cnt : ARRAY[0..24] OF USINT; (*Counter (-)*)
        rFenst2_Vect : ARRAY[0..24] OF REAL; (*Mechanical noise of valid cylinders (mV)*)
        bValidCyl : ARRAY[0..24] OF BOOL; (*Vector indicating valid cylinders for monitoring (-)*)
        rFiltTau_Lim : REAL; (*Parameter limitation: Mechanical noise filter factor (-)*)
        rFiltGain_Lim : REAL; (*Parameter limitation: Mechanical noise filter gain (-)*)
        rMargTexhAct_Lim : REAL; (*Parameter limitation: Threshold where Texh Monitoring uses narrow margin (-)*)
        rOffMeNoi_Lim : REAL; (*Parameter limitation: Mechanical noise filter offset factor (-)*)
        rFenst2LiMx_Lim : REAL; (*Parameter limitation: Max Limit for Mechanical Noise detection (mV)*)
        rFenst2LiMn_Lim : REAL; (*Parameter limitation: Limit for measuring signal failure (mV)*)
        uAdapLim_MeNoi_Cyl : ARRAY[0..24] OF REAL; (*Cylinder individual adaptive mechanical noise limit (mV)*)
        uAdapLim_Marg : REAL; (*Mechanical noise average based limit (mV)*)
    END_STRUCT;

   tMeNoiAL_IN : STRUCT
        ucNumCyl : USINT; (*Total number of cylinders (-)*)
        bKnockSig : ARRAY[0..24] OF BOOL; (*Measurement signal error (-)*)
        bGCB_On_TC2_Di : BOOL; (*GCB closed (-)*)
        uFenst2 : ARRAY[0..24] OF UINT; (*Mechanical noise per cylinder (mV)*)
    END_STRUCT;

   tMeNoiAL_OUT : STRUCT
        bTExh_Mon_UseNarrowWindow : ARRAY[0..24] OF BOOL; (*narrower threshold activation for exhaust temperature monitoring (-)*)
        bValve : ARRAY[0..24] OF BOOL; (*mech noise cyl individual alarm activation (-)*)
        uFenst2_Av : UINT; (*mechanical noise average (-)*)
        uFenst2_Mx : UINT; (*maximum mechanical noise (-)*)
        uFenst2_Mn : UINT; (*minimum mechanical noise (-)*)
    END_STRUCT;

   tMeNoiAL_PARA : STRUCT
        rFenst2LiMx : REAL; (*Max Limit for Mechanical Noise detection (mV)*)
        rFenst2LiMn : REAL; (*Limit for measuring signal failure (mV)*)
        rFiltTau_MeNoi : REAL; (*Mechanical Noise filter factor (-)*)
        rMargTExh_Active : REAL; (*Threshold where Texh Monitoring uses narrow margin (-)*)
        bMeNoi_Active : BOOL; (*Mechanical Noise Adaptive Limit Active (-)*)
    END_STRUCT;
END_TYPE
TYPE
BlockIO_MeNoiAL : STRUCT
	BusInput : tMeNoiAL_IN;
	BusInput1 : tMeNoiAL_PARA;
	UnitDelay : UDINT;
END_STRUCT;
D_Work_MeNoiAL : STRUCT
	Delay_DSTATE : ARRAY[0..24] OF REAL;
	DiscreteTimeIntegrator_DSTATE : ARRAY[0..24] OF REAL;
	UnitDelay_DSTATE : UDINT;
	Delay_DSTATE_c : ARRAY[0..24] OF USINT;
	DiscreteTimeIntegrator_PrevRese : SINT;
	DiscreteTimeIntegrator_IC_LOADI : USINT;
END_STRUCT;
ConstBlockIO_MeNoiAL : STRUCT
	DataTypeConversion : ARRAY[0..24] OF REAL;
END_STRUCT;
ExternalInputs_MeNoiAL : STRUCT
	In_MeNnoiAL : tMeNoiAL_IN;
	Para_MeNoiAL : tMeNoiAL_PARA;
END_STRUCT;
ExternalOutputs_MeNoiAL : STRUCT
	Out_MeNoiAL : tMeNoiAL_OUT;
	Dbg_MeNoiAL : tMeNoiAL_DBG;
END_STRUCT;
END_TYPE
```
